      L     #Offset;
      SLD   3;
      LAR2;  // Recupero que offset tiene la String

// --- Ya esta convertido el Valor a ASCI - Fin Patin
CodigoPatin_NUUT_EventosUT:NOP   0;





////////////////////////////////////////////////////////////////////////////////
// --- Atributo de ETIQUETA (Si es necesario) --- Router
      SET;  // Tiene Etiqueta
      AN    "DB850_DefinicionMesas".Mesa[#NumMesa].AtributosGalibo_DeEvento.EtiquetaRouter;
      JC    FinEtiquetaRouter_NUUT_EventoUT;

      OPN   DB [#DBEventos];
      L     '[';  // Evento - Atributo Etiqueta '[SSCC]'
      T     DBB [AR2, P#0.0];
      L     'SSCC';
      T     DBD [AR2, P#1.0];
      L     ']';
      T     DBB [AR2, P#5.0];
      +AR2  P#6.0;

      L     "DB814_UTs_Etiqueta".UT[#NumeroUT].EtiquetaRouter;
      T     #Valor;

// --- Convertir Valor a ASCII -  Etiqueta de Router
      TAR2;
      SRD   3;
      T     #NumBytes;  // Miro que offset tiene la String

      CALL  "FC893_Obtener_StringDelAtributo"
      ( DB_String := #NumDBEventos,
        OffsetIni := #NumBytes,
        Valor     := #Valor,
        OffsetFin := #Offset
      );  // Llamo a ObtenerStrinAtributo

      L     #Offset;
      SLD   3;
      LAR2;  // Recupero que offset tiene la String

// --- Ya esta convertido el Valor a ASCI - Fin Etiqueta de Router
FinEtiquetaRouter_NUUT_EventoUT:NOP   0;





////////////////////////////////////////////////////////////////////////////////
// --- Atributo de ETIQUETA (Si es necesario) ---  STRING
      SET;  // Tiene Etiqueta
      AN    "DB850_DefinicionMesas".Mesa[#NumMesa].AtributosGalibo_DeEvento.EtiquetaString;
      JC    FinEtiquetaString_NUUT_EventoUT;

      OPN   DB [#DBEventos];
      L     '[';  // Evento - Atributo Etiqueta '[SSCC]'
      T     DBB [AR2, P#0.0];
      L     'SSCC';
      T     DBD [AR2, P#1.0];
      L     ']';
      T     DBB [AR2, P#5.0];
      +AR2  P#6.0;

      L     2;  // Puntero a la Etiqueta
      T     #IndiceEtiqueta;

BucleEtiquetastring_NUUT_EventoUT:NOP   0;
      L     "DB814_UTs_Etiqueta".UT[#NumeroUT].Etiqueta[#IndiceEtiqueta];
      T     #Valor;  // Recoge el caracter de la Etiqueta

      L     #Valor;
      L     0;
      ==D;  // Es Final de Etiqueta?
      JC    FinEtiquetaString_NUUT_EventoUT;

      OPN   DB [#DBEventos];
      L     #Valor;
      T     DBB [AR2, P#0.0];

      L     #IndiceEtiqueta;  // Siguiente Caracter
      L     1;
      +I;
      T     #IndiceEtiqueta;
      +AR2  P#1.0;

      JU    BucleEtiquetastring_NUUT_EventoUT;

FinEtiquetaString_NUUT_EventoUT:NOP   0;


////////////////////////////////////////////////////////////////////////////////-
// --- Final del Formato del Evento ---

      OPN   DB [#DBEventos];  // DB de Eventos Generados (A Emitir)
      L     '}';  // Fin de Evento '}'
      T     DBB [AR2, P#0.0];
      +AR2  P#1.0;

////////////////////////////////////////////////////////////////////////////////
////////////////////////////////////////////////////////////////////////////////
////////////////////////////////////////////////////////////////////////////////
////////////////////////////////////////////////////////////////////////////////
// Dar por formateado el Evento
// Borrar la UT de la Base de datos (Por Presencias Multiples de las Mesas)
// Solo no se borra cuando la Mesa es Remota, no debe ni entrar aqui.

      CALL  "FC722_EliminarUT_DeMesa"
      ( NumeroUT := #NumeroUT
      );

      JU    FinBucles_EventosUT;

// Fin del Evento NUUT
////////////////////////////////////////////////////////////////////////////////
////////////////////////////////////////////////////////////////////////////////
////////////////////////////////////////////////////////////////////////////////
////////////////////////////////////////////////////////////////////////////////



NETWORK
TITLE = ---- Evento de UT - Refresco de Datos de la UT -- DATO
GenerarEvento_DATO_EventoUT:NOP   0;

////////////////////////////////////////////////////////////////////////////////
////////////////////////////////////////////////////////////////////////////////
////////////////////////////////////////////////////////////////////////////////
////////////////////////////////////////////////////////////////////////////////
// -- Formateo del Evento DATO - Refresco de Datos de la UT

      L     #P_Eventos;
      LAR2;  // Puntero al DB de Eventos Generados

      TAR2;  // Mirar si es el primer evento de la lista
      L     0;
      ==I;
      JC    InicioBuffer_DATO_EventosUT;  // Es el primero

      OPN   DB [#DBEventos];  // Hay que añadir si no es el primer evento
      L     ',';  // Separador entre eventos ','
      T     DBB [AR2, P#0.0];
      +AR2  P#1.0;

InicioBuffer_DATO_EventosUT:NOP   0;
      OPN   DB [#DBEventos];  // DB de Eventos Generados (A Emitir)
      L     '{';  // Inicio de Evento '{'
      T     DBB [AR2, P#0.0];
      +AR2  P#1.0;

      L     'DATO';  // Evento 'DATO'
      T     DBD [AR2, P#0.0];
      +AR2  P#4.0;


////////////////////////////////////////////////////////////////////////////////
      L     '[';  // Evento - Atributo Mckey '[MCKY]'
      T     DBB [AR2, P#0.0];
      L     'MCKY';
      T     DBD [AR2, P#1.0];
      L     ']';
      T     DBB [AR2, P#5.0];
      +AR2  P#6.0;

      L     "DB812_UTs_Control".UT[#NumeroUT].Mckey;
      T     #Valor;

// --- Convertir Valor a ASCII - Mckey
      TAR2;
      SRD   3;
      T     #NumBytes;  // Miro que offset tiene la String

      CALL  "FC893_Obtener_StringDelAtributo"
      ( DB_String := #NumDBEventos,
        OffsetIni := #NumBytes,
        Valor     := #Valor,
        OffsetFin := #Offset
      );  // Llamo a ObtenerStrinAtributo

      L     #Offset;
      SLD   3;
      LAR2;  // Recupero que offset tiene la String

// --- Ya esta convertido el Valor a ASCI - Fin Mckey


////////////////////////////////////////////////////////////////////////////////
      OPN   DB [#DBEventos];
      L     '[';  // Evento - Atributo Mesa Actual '[MESA]'
      T     DBB [AR2, P#0.0];
      L     'MESA';
      T     DBD [AR2, P#1.0];
      L     ']';
      T     DBB [AR2, P#5.0];
      +AR2  P#6.0;

      L     "DB812_UTs_Control".UT[#NumeroUT].MesaActual;
      T     #Valor;

// --- Convertir Valor a ASCII -  Mesa Actual
      TAR2;
      SRD   3;
      T     #NumBytes;  // Miro que offset tiene la String

      CALL  "FC893_Obtener_StringDelAtributo"
      ( DB_String := #NumDBEventos,
        OffsetIni := #NumBytes,
        Valor     := #Valor,
        OffsetFin := #Offset
      );  // Llamo a ObtenerStrinAtributo

      L     #Offset;
      SLD   3;
      LAR2;  // Recupero que offset tiene la String

// --- Ya esta convertido el Valor a ASCI - Fin Mesa Actual


////////////////////////////////////////////////////////////////////////////////
////////////////////////////////////////////////////////////////////////////////
////////////////////////////////////////////////////////////////////////////////
////////////////////////////////////////////////////////////////////////////////
// --- Caracteristicas de la UT a Emitir


////////////////////////////////////////////////////////////////////////////////
// --- Atributo de ALTURA COTA (Si es necesario) ---
      SET;  // Tiene Cota de Altura ?
      AN    "DB850_DefinicionMesas".Mesa[#NumMesa].AtributosGalibo_DeEvento.Cota_Altura;
      JC    CotaAltura_DATO_EventoUT;

      L     "DB815_UTs_Datos".UT[#NumeroUT].CotaAltura;
      T     #Valor;

      OPN   DB [#DBEventos];
      L     '[';  // Evento - Atributo Altura Cota '[COTA]'
      T     DBB [AR2, P#0.0];
      L     'COTA';
      T     DBD [AR2, P#1.0];
      L     ']';
      T     DBB [AR2, P#5.0];
      +AR2  P#6.0;

// --- Convertir Valor a ASCII -  Altura Cota
      TAR2;
      SRD   3;
      T     #NumBytes;  // Miro que offset tiene la String

      CALL  "FC893_Obtener_StringDelAtributo"
      ( DB_String := #NumDBEventos,
        OffsetIni := #NumBytes,
        Valor     := #Valor,
        OffsetFin := #Offset
      );  // Llamo a ObtenerStrinAtributo

      L     #Offset;
      SLD   3;
      LAR2;  // Recupero que offset tiene la String

// --- Ya esta convertido el Valor a ASCI - Fin Altura Cota
CotaAltura_DATO_EventoUT:NOP   0;


////////////////////////////////////////////////////////////////////////////////
////////////////////////////////////////////////////////////////////////////////
////////////////////////////////////////////////////////////////////////////////
////////////////////////////////////////////////////////////////////////////////
// --- Atributo de GALIBO (Si es necesario) ---
      SET;  // Tiene Altura ?
      AN    "DB850_DefinicionMesas".Mesa[#NumMesa].AtributosGalibo_DeEvento.Altura;
      JC    CodigoAltura_DATO_EventoUT;

      OPN   DB [#DBEventos];
      L     '[';  // Evento - Atributo Galibo Altura '[ALTO]'
      T     DBB [AR2, P#0.0];
      L     'ALTO';
      T     DBD [AR2, P#1.0];
      L     ']';
      T     DBB [AR2, P#5.0];
      +AR2  P#6.0;

      L     "DB815_UTs_Datos".UT[#NumeroUT].GaliboAltura;
      T     #Valor;

// --- Convertir Valor a ASCII -  Alto
      TAR2;
      SRD   3;
      T     #NumBytes;  // Miro que offset tiene la String

      CALL  "FC893_Obtener_StringDelAtributo"
      ( DB_String := #NumDBEventos,
        OffsetIni := #NumBytes,
        Valor     := #Valor,
        OffsetFin := #Offset
      );  // Llamo a ObtenerStrinAtributo

      L     #Offset;
      SLD   3;
      LAR2;  // Recupero que offset tiene la String


// nieves inicio modificación emisión atributo VACI

//Comprobar si tenemos que emitir el evento

      SET;
      L     "DB815_UTs_Datos".UT[#NumeroUT].GaliboVacia;
      L     0;
      ==I;
      JC    CodigoAltura_DATO_EventoUT;

      OPN   DB [#DBEventos];
      L     '[';  // Evento - Atributo Galibo Altura '[ALTO]'
      T     DBB [AR2, P#0.0];
      L     'VACI';
      T     DBD [AR2, P#1.0];
      L     ']';
      T     DBB [AR2, P#5.0];
      +AR2  P#6.0;

      L     "DB815_UTs_Datos".UT[#NumeroUT].GaliboVacia;
      L     1;
      -I;
      T     #Valor;

// --- Convertir Valor a ASCII -  VACIO
      TAR2;
      SRD   3;
      T     #NumBytes;  // Miro que offset tiene la String

      CALL  "FC893_Obtener_StringDelAtributo"
      ( DB_String := #NumDBEventos,
        OffsetIni := #NumBytes,
        Valor     := #Valor,
        OffsetFin := #Offset
      );  // Llamo a ObtenerStrinAtributo


      L     #Offset;
      SLD   3;
      LAR2;  // Recupero que offset tiene la String


// fin modificación atributo VACI

// --- Ya esta convertido el Valor a ASCI - Fin Alto
CodigoAltura_DATO_EventoUT:NOP   0;


////////////////////////////////////////////////////////////////////////////////
      SET;  // Tien Anchura ?
      AN    "DB850_DefinicionMesas".Mesa[#NumMesa].AtributosGalibo_DeEvento.Anchura;
      JC    CodigAnchura_DATO_EventoUT;

      OPN   DB [#DBEventos];
      L     '[';  // Evento - Atributo Galibo Anchura '[ANCH]'
      T     DBB [AR2, P#0.0];
      L     'ANCH';
      T     DBD [AR2, P#1.0];
      L     ']';
      T     DBB [AR2, P#5.0];
      +AR2  P#6.0;

      L     "DB815_UTs_Datos".UT[#NumeroUT].GaliboAnchura;
      T     #Valor;

// --- Convertir Valor a ASCII -  Anchura
      TAR2;
      SRD   3;
      T     #NumBytes;  // Miro que offset tiene la String

      CALL  "FC893_Obtener_StringDelAtributo"
      ( DB_String := #NumDBEventos,
        OffsetIni := #NumBytes,
        Valor     := #Valor,
        OffsetFin := #Offset
      );  // Llamo a ObtenerStrinAtributo

      L     #Offset;
      SLD   3;
      LAR2;  // Recupero que offset tiene la String

// --- Ya esta convertido el Valor a ASCI - Fin Anchura
CodigAnchura_DATO_EventoUT:NOP   0;


////////////////////////////////////////////////////////////////////////////////
      SET;  // Tiene Profundidad ?
      AN    "DB850_DefinicionMesas".Mesa[#NumMesa].AtributosGalibo_DeEvento.Profundidad;
      JC    CodigLargura_DATO_EventoUT;

      OPN   DB [#DBEventos];
      L     '[';  // Evento - Atributo Galibo Profuncidad '[PROF]'
      T     DBB [AR2, P#0.0];
      L     'PROF';
      T     DBD [AR2, P#1.0];
      L     ']';
      T     DBB [AR2, P#5.0];
      +AR2  P#6.0;

      L     "DB815_UTs_Datos".UT[#NumeroUT].GaliboProfundidad;
      T     #Valor;

// --- Convertir Valor a ASCII -  Largura
      TAR2;
      SRD   3;
      T     #NumBytes;  // Miro que offset tiene la String

      CALL  "FC893_Obtener_StringDelAtributo"
      ( DB_String := #NumDBEventos,
        OffsetIni := #NumBytes,
        Valor     := #Valor,
        OffsetFin := #Offset
      );  // Llamo a ObtenerStrinAtributo

      L     #Offset;
      SLD   3;
      LAR2;  // Recupero que offset tiene la String

// --- Ya esta convertido el Valor a ASCI - Fin Largura
CodigLargura_DATO_EventoUT:NOP   0;


////////////////////////////////////////////////////////////////////////////////
      SET;  // Tiene Remontado ?
      AN    "DB850_DefinicionMesas".Mesa[#NumMesa].AtributosGalibo_DeEvento.Remontado;
      JC    CodigRemontado_DATO_EventoUT;

      OPN   DB [#DBEventos];
      L     '[';  // Evento - Atributo Galibo Remontada '[REMO]'
      T     DBB [AR2, P#0.0];
      L     'REMO';
      T     DBD [AR2, P#1.0];
      L     ']';
      T     DBB [AR2, P#5.0];
      +AR2  P#6.0;

      L     "DB815_UTs_Datos".UT[#NumeroUT].GaliboRemontada;
      L     1;
      -I;
      L     W#16#30;
      +I;
      OPN   DB [#DBEventos];
      T     DBB [AR2, P#0.0];
      +AR2  P#1.0;

CodigRemontado_DATO_EventoUT:NOP   0;


////////////////////////////////////////////////////////////////////////////////
// --- Atributo de PESO (Si es necesario) ---
      SET;  // Tiene Peso ?
      AN    "DB850_DefinicionMesas".Mesa[#NumMesa].AtributosGalibo_DeEvento.Peso;
      JC    Peso_DATO_EventoUT;

      OPN   DB [#DBEventos];
      L     '[';  // Evento - Atributo Peso '[PESO]'
      T     DBB [AR2, P#0.0];
      L     'PESO';
      T     DBD [AR2, P#1.0];
      L     ']';
      T     DBB [AR2, P#5.0];
      +AR2  P#6.0;

      L     "DB815_UTs_Datos".UT[#NumeroUT].Peso;
      T     #Valor;

// --- Convertir Valor a ASCII -  Peso
      TAR2;
      SRD   3;
      T     #NumBytes;  // Miro que offset tiene la String

      CALL  "FC893_Obtener_StringDelAtributo"
      ( DB_String := #NumDBEventos,
        OffsetIni := #NumBytes,
        Valor     := #Valor,
        OffsetFin := #Offset
      );  // Llamo a ObtenerStrinAtributo

      L     #Offset;
      SLD   3;
      LAR2;  // Recupero que offset tiene la String

// --- Ya esta convertido el Valor a ASCI - Fin Peso
Peso_DATO_EventoUT:NOP   0;


////////////////////////////////////////////////////////////////////////////////
// --- Atributo de ANCHURA COTA (Si es necesario) ---
      SET;  // Tiene Cota de Anchura ?
      AN    "DB850_DefinicionMesas".Mesa[#NumMesa].AtributosGalibo_DeEvento.Cota_Anchura;
      JC    CotaAnchura_DATO_EventoUT;

      L     "DB815_UTs_Datos".UT[#NumeroUT].CotaAnchura;
      T     #Valor;

      OPN   DB [#DBEventos];
      L     '[';  // Evento - Atributo Anchura Cota '[COTW]'
      T     DBB [AR2, P#0.0];
      L     'COTW';
      T     DBD [AR2, P#1.0];
      L     ']';
      T     DBB [AR2, P#5.0];
      +AR2  P#6.0;

// --- Convertir Valor a ASCII -  Anchura Cota
      TAR2;
      SRD   3;
      T     #NumBytes;  // Miro que offset tiene la String

      CALL  "FC893_Obtener_StringDelAtributo"
      ( DB_String := #NumDBEventos,
        OffsetIni := #NumBytes,
        Valor     := #Valor,
        OffsetFin := #Offset
      );  // Llamo a ObtenerStrinAtributo

      L     #Offset;
      SLD   3;
      LAR2;  // Recupero que offset tiene la String

// --- Ya esta convertido el Valor a ASCI - Fin Anchura Cota
CotaAnchura_DATO_EventoUT:NOP   0;


////////////////////////////////////////////////////////////////////////////////
// --- Atributo de LARGURA COTA (Si es necesario) ---
      SET;  // Tiene Cota de Profundidad ?
      AN    "DB850_DefinicionMesas".Mesa[#NumMesa].AtributosGalibo_DeEvento.Cota_Profundidad;
      JC    CotaLargura_DATO_EventoUT;

      L     "DB815_UTs_Datos".UT[#NumeroUT].CotaProfundidad;
      T     #Valor;

      OPN   DB [#DBEventos];
      L     '[';  // Evento - Atributo Largura Cota '[COTL]'
      T     DBB [AR2, P#0.0];
      L     'COTL';
      T     DBD [AR2, P#1.0];
      L     ']';
      T     DBB [AR2, P#5.0];
      +AR2  P#6.0;

// --- Convertir Valor a ASCII -  Largura Cota
      TAR2;
      SRD   3;
      T     #NumBytes;  // Miro que offset tiene la String

      CALL  "FC893_Obtener_StringDelAtributo"
      ( DB_String := #NumDBEventos,
        OffsetIni := #NumBytes,
        Valor     := #Valor,
        OffsetFin := #Offset
      );  // Llamo a ObtenerStrinAtributo

      L     #Offset;
      SLD   3;
      LAR2;  // Recupero que offset tiene la String

// --- Ya esta convertido el Valor a ASCI - Fin Largura Cota
CotaLargura_DATO_EventoUT:NOP   0;


////////////////////////////////////////////////////////////////////////////////
////////////////////////////////////////////////////////////////////////////////
////////////////////////////////////////////////////////////////////////////////
// --- Atributo de TIPO, HUECO y TACO (Si es necesario) ---
      SET;  // Tiene Taco ?
      AN    "DB850_DefinicionMesas".Mesa[#NumMesa].AtributosGalibo_DeEvento.Taco;
      JC    CodigoTaco_DATO_EventoUT;

      OPN   DB [#DBEventos];
      L     '[';  // Evento - Atributo Galibo Taco '[TACO]'
      T     DBB [AR2, P#0.0];
      L     'TACO';
      T     DBD [AR2, P#1.0];
      L     ']';
      T     DBB [AR2, P#5.0];
      +AR2  P#6.0;

      L     "DB815_UTs_Datos".UT[#NumeroUT].GaliboTaco;
      T     #Valor;

// --- Convertir Valor a ASCII -  Taco
      TAR2;
      SRD   3;
      T     #NumBytes;  // Miro que offset tiene la String

      CALL  "FC893_Obtener_StringDelAtributo"
      ( DB_String := #NumDBEventos,
        OffsetIni := #NumBytes,
        Valor     := #Valor,
        OffsetFin := #Offset
      );  // Llamo a ObtenerStrinAtributo

      L     #Offset;
      SLD   3;
      LAR2;  // Recupero que offset tiene la String

// --- Ya esta convertido el Valor a ASCI - Fin Taco
CodigoTaco_DATO_EventoUT:NOP   0;


////////////////////////////////////////////////////////////////////////////////
      SET;  // Tiene Hueco ?
      AN    "DB850_DefinicionMesas".Mesa[#NumMesa].AtributosGalibo_DeEvento.Hueco;
      JC    CodigoHueco_DATO_EventoUT;

      OPN   DB [#DBEventos];
      L     '[';  // Evento - Atributo Galibo Hueco '[HUEC]'
      T     DBB [AR2, P#0.0];
      L     'HUEC';
      T     DBD [AR2, P#1.0];
      L     ']';
      T     DBB [AR2, P#5.0];
      +AR2  P#6.0;

      L     "DB815_UTs_Datos".UT[#NumeroUT].GaliboHueco;
      T     #Valor;

// --- Convertir Valor a ASCII -  Hueco
      TAR2;
      SRD   3;
      T     #NumBytes;  // Miro que offset tiene la String

      CALL  "FC893_Obtener_StringDelAtributo"
      ( DB_String := #NumDBEventos,
        OffsetIni := #NumBytes,
        Valor     := #Valor,
        OffsetFin := #Offset
      );  // Llamo a ObtenerStrinAtributo

      L     #Offset;
      SLD   3;
      LAR2;  // Recupero que offset tiene la String

// --- Ya esta convertido el Valor a ASCI - Fin Hueco
CodigoHueco_DATO_EventoUT:NOP   0;


////////////////////////////////////////////////////////////////////////////////
      SET;  // Tiene Hueco_R
      AN    "DB850_DefinicionMesas".Mesa[#NumMesa].AtributosGalibo_DeEvento.HuecoRemontado;
      JC    CodigoHuecoR_DATO_EventoUT;

      OPN   DB [#DBEventos];
      L     '[';  // Evento - Atributo Galibo Hueco '[HUEC]'
      T     DBB [AR2, P#0.0];
      L     'HUER';
      T     DBD [AR2, P#1.0];
      L     ']';
      T     DBB [AR2, P#5.0];
      +AR2  P#6.0;

      L     "DB815_UTs_Datos".UT[#NumeroUT].GaliboHuecoRemontado;
      T     #Valor;

// --- Convertir Valor a ASCII -  Hueco R
      TAR2;
      SRD   3;
      T     #NumBytes;  // Miro que offset tiene la String

      CALL  "FC893_Obtener_StringDelAtributo"
      ( DB_String := #NumDBEventos,
        OffsetIni := #NumBytes,
        Valor     := #Valor,
        OffsetFin := #Offset
      );  // Llamo a ObtenerStrinAtributo

      L     #Offset;
      SLD   3;
      LAR2;  // Recupero que offset tiene la String

// --- Ya esta convertido el Valor a ASCI - Fin Hueco R
CodigoHuecoR_DATO_EventoUT:NOP   0;


////////////////////////////////////////////////////////////////////////////////
      SET;  // Tiene Tipo ?
      AN    "DB850_DefinicionMesas".Mesa[#NumMesa].AtributosGalibo_DeEvento.Tipo;
      JC    CodigoTipo_DATO_EventoUT;

      OPN   DB [#DBEventos];
      L     '[';  // Evento - Atributo Galibo Hueco '[HUEC]'
      T     DBB [AR2, P#0.0];
      L     'TIPO';
      T     DBD [AR2, P#1.0];
      L     ']';
      T     DBB [AR2, P#5.0];
      +AR2  P#6.0;

      L     "DB815_UTs_Datos".UT[#NumeroUT].GaliboTipoCarga;
      L     W#16#F;
      <>I;
      JC    CodigoTipoExiste_DATO_EventoUT;

      OPN   DB [#DBEventos];
      L     'ERRO';
      T     DBD [AR2, P#0.0];
      +AR2  P#4.0;

      JU    CodigoTipo_DATO_EventoUT;

CodigoTipoExiste_DATO_EventoUT:NOP   0;
      L     "DB815_UTs_Datos".UT[#NumeroUT].GaliboTipoCarga;
      L     3000;
      +I;
      T     #Convertir;
      CALL  "FC895_Obtener_EtiquetaDeValor"
      ( ValorEvento    := #Convertir,
        EtiquetaEvento := #Conversion
      );

      OPN   DB [#DBEventos];
      L     #Conversion;
      T     DBD [AR2, P#0.0];
      +AR2  P#4.0;

CodigoTipo_DATO_EventoUT:NOP   0;


////////////////////////////////////////////////////////////////////////////////
////////////////////////////////////////////////////////////////////////////////
////////////////////////////////////////////////////////////////////////////////
// --- Atributo de COLOR (Si es necesario) ---
      SET;  // Tiene Color ?
      AN    "DB850_DefinicionMesas".Mesa[#NumMesa].AtributosGalibo_DeEvento.Color;
      JC    CodigoColor_DATO_EventoUT;

      OPN   DB [#DBEventos];
      L     '[';  // Evento - Atributo Galibo Hueco '[HUEC]'
      T     DBB [AR2, P#0.0];
      L     'COLO';
      T     DBD [AR2, P#1.0];
      L     ']';
      T     DBB [AR2, P#5.0];
      +AR2  P#6.0;

      L     "DB815_UTs_Datos".UT[#NumeroUT].GaliboColor;
      L     W#16#F;
      <>I;
      JC    CodigoColorExiste_DATO_EventoUT;

      OPN   DB [#DBEventos];
      L     'ERRO';
      T     DBD [AR2, P#0.0];
      +AR2  P#4.0;

      JU    CodigoColor_DATO_EventoUT;

CodigoColorExiste_DATO_EventoUT:NOP   0;
      L     "DB815_UTs_Datos".UT[#NumeroUT].GaliboColor;
      L     3100;
      +I;
      T     #Convertir;
      CALL  "FC895_Obtener_EtiquetaDeValor"
      ( ValorEvento    := #Convertir,
        EtiquetaEvento := #Conversion
      );

      OPN   DB [#DBEventos];
      L     #Conversion;
      T     DBD [AR2, P#0.0];
      +AR2  P#4.0;

CodigoColor_DATO_EventoUT:NOP   0;

////////////////////////////////////////////////////////////////////////////////
      SET;  // Tiene Patin ?
      AN    "DB850_DefinicionMesas".Mesa[#NumMesa].AtributosGalibo_DeEvento.Patin;
      JC    CodigoPatin_DATO_EventoUT;

      OPN   DB [#DBEventos];
      L     '[';  // Evento - Atributo Galibo Patin '[PATI]'
      T     DBB [AR2, P#0.0];
      L     'PATI';
      T     DBD [AR2, P#1.0];
      L     ']';
      T     DBB [AR2, P#5.0];
      +AR2  P#6.0;

      L     "DB815_UTs_Datos".UT[#NumeroUT].GaliboPatin;
      T     #Valor;

// --- Convertir Valor a ASCII -  Patin
      TAR2;
      SRD   3;
      T     #NumBytes;  // Miro que offset tiene la String

      CALL  "FC893_Obtener_StringDelAtributo"
      ( DB_String := #NumDBEventos,
        OffsetIni := #NumBytes,
        Valor     := #Valor,
        OffsetFin := #Offset
      );  // Llamo a ObtenerStrinAtributo

      L     #Offset;
      SLD   3;
      LAR2;  // Recupero que offset tiene la String

// --- Ya esta convertido el Valor a ASCI - Fin Patin
CodigoPatin_DATO_EventoUT:NOP   0;



////////////////////////////////////////////////////////////////////////////////
// --- Atributo de ETIQUETA (Si es necesario) --- Router
      SET;  // Tiene Etiqueta ?
      AN    "DB850_DefinicionMesas".Mesa[#NumMesa].AtributosGalibo_DeEvento.EtiquetaRouter;
      JC    FinEtiquetaRouter_DATO_EventoUT;

      OPN   DB [#DBEventos];
      L     '[';  // Evento - Atributo Etiqueta '[SSCC]'
      T     DBB [AR2, P#0.0];
      L     'SSCC';
      T     DBD [AR2, P#1.0];
      L     ']';
      T     DBB [AR2, P#5.0];
      +AR2  P#6.0;

      L     0;  // Puntero a la Etiqueta
      T     #IndiceEtiqueta;

      L     "DB814_UTs_Etiqueta".UT[#NumeroUT].EtiquetaRouter;
      T     #Valor;  // Recoge el caracter de la Etiqueta

// --- Convertir Valor a ASCII -  Etiqueta Router
      TAR2;
      SRD   3;
      T     #NumBytes;  // Miro que offset tiene la String

      CALL  "FC893_Obtener_StringDelAtributo"
      ( DB_String := #NumDBEventos,
        OffsetIni := #NumBytes,
        Valor     := #Valor,
        OffsetFin := #Offset
      );  // Llamo a ObtenerStrinAtributo

      L     #Offset;
      SLD   3;
      LAR2;  // Recupero que offset tiene la String

// --- Ya esta convertido el Valor a ASCI - Fin Etiqueta Router
FinEtiquetaRouter_DATO_EventoUT:NOP   0;







////////////////////////////////////////////////////////////////////////////////
// --- Atributo de ETIQUETA (Si es necesario) --- STRING
      SET;  // Tiene Etiqueta ?
      AN    "DB850_DefinicionMesas".Mesa[#NumMesa].AtributosGalibo_DeEvento.EtiquetaString;
      JC    FinEtiquetaString_DATO_EventoUT;

      OPN   DB [#DBEventos];
      L     '[';  // Evento - Atributo Etiqueta '[SSCC]'
      T     DBB [AR2, P#0.0];
      L     'SSCC';
      T     DBD [AR2, P#1.0];
      L     ']';
      T     DBB [AR2, P#5.0];
      +AR2  P#6.0;

      L     2;  // Puntero a la Etiqueta
      T     #IndiceEtiqueta;

BucleEtiquetaString_DATO_EventoUT:NOP   0;
      L     "DB814_UTs_Etiqueta".UT[#NumeroUT].Etiqueta[#IndiceEtiqueta];
      T     #Valor;  // Recoge el caracter de la Etiqueta

      L     #Valor;
      L     0;
      ==I;
      JC    FinEtiquetaString_DATO_EventoUT;  // Es Final de Etiqueta?

      OPN   DB [#DBEventos];
      L     #Valor;
      T     DBB [AR2, P#0.0];

      L     #IndiceEtiqueta;  // Siguiente Caracter
      L     1;
      +I;
      T     #IndiceEtiqueta;
      +AR2  P#1.0;
      JU    BucleEtiquetaString_DATO_EventoUT;

FinEtiquetaString_DATO_EventoUT:NOP   0;





////////////////////////////////////////////////////////////////////////////////
// --- Final del Formato del Evento ---

      OPN   DB [#DBEventos];  // DB de Eventos Generados (A Emitir)
      L     '}';  // Fin de Evento '}'
      T     DBB [AR2, P#0.0];
      +AR2  P#1.0;


////////////////////////////////////////////////////////////////////////////////
////////////////////////////////////////////////////////////////////////////////
////////////////////////////////////////////////////////////////////////////////
////////////////////////////////////////////////////////////////////////////////
// Dar por formateado el Evento

      L     0;  // 0 - Dar por Tratado
      T     "DB812_UTs_Control".UT[#NumeroUT].EstadoEventoAGenerar;

////////////////////////////////////////////////////////////////////////////////
/// Hay que Pedir Datos
      SET;
      AN    "DB812_UTs_Control".UT[#NumeroUT].AtributosDeLaUT.PeticionDeDatos;
      JC    NoPedirDatos_DATO_EventosUT;

      L     141;
      T     "DB812_UTs_Control".UT[#NumeroUT].EstadoEventoAGenerar;

NoPedirDatos_DATO_EventosUT:NOP   0;


////////////////////////////////////////////////////////////////////////////////
      JU    FinBucles_EventosUT;


// Fin del formateo del Evento DATO
////////////////////////////////////////////////////////////////////////////////
////////////////////////////////////////////////////////////////////////////////
////////////////////////////////////////////////////////////////////////////////
////////////////////////////////////////////////////////////////////////////////



NETWORK
TITLE = ---- Evento de UT - Peticion de Datos de la UT - DAT?
GenerarEvento_DAT_EventosUT:NOP   0;

////////////////////////////////////////////////////////////////////////////////
////////////////////////////////////////////////////////////////////////////////
////////////////////////////////////////////////////////////////////////////////
// -- Formateo del Evento DAT? - Peticion de Datos para la UT
// -- Hay que poner que campo?       ¡¡¡ OJO !!!

      L     #P_Eventos;
      LAR2;  // Puntero al DB de Eventos Generados

      TAR2;  // Mirar si es el primer evento de la lista
      L     0;
      ==I;
      JC    InicioBuffer_DAT_EventosUT;  // Es el primero

      OPN   DB [#DBEventos];  // Hay que añadir si no es el primer evento
      L     ',';  // Separador entre eventos ','
      T     DBB [AR2, P#0.0];
      +AR2  P#1.0;

InicioBuffer_DAT_EventosUT:NOP   0;
      OPN   DB [#DBEventos];  // DB de Eventos Generados (A Emitir)
      L     '{';  // Inicio de Evento '{'
      T     DBB [AR2, P#0.0];
      +AR2  P#1.0;

      L     'DAT?';  // Evento 'DAT?'
      T     DBD [AR2, P#0.0];
      +AR2  P#4.0;


////////////////////////////////////////////////////////////////////////////////
      L     '[';  // Evento - Atributo Mckey '[MCKY]'
      T     DBB [AR2, P#0.0];
      L     'MCKY';
      T     DBD [AR2, P#1.0];
      L     ']';
      T     DBB [AR2, P#5.0];
      +AR2  P#6.0;

      L     "DB812_UTs_Control".UT[#NumeroUT].Mckey;
      T     #Valor;

// --- Convertir Valor a ASCII - Mckey
      TAR2;
      SRD   3;
      T     #NumBytes;  // Miro que offset tiene la String

      CALL  "FC893_Obtener_StringDelAtributo"
      ( DB_String := #NumDBEventos,
        OffsetIni := #NumBytes,
        Valor     := #Valor,
        OffsetFin := #Offset
      );  // Llamo a ObtenerStrinAtributo

      L     #Offset;
      SLD   3;
      LAR2;  // Recupero que offset tiene la String

// --- Ya esta convertido el Valor a ASCI - Fin Mckey


////////////////////////////////////////////////////////////////////////////////
      OPN   DB [#DBEventos];
      L     '[';  // Evento - Atributo Mesa Actual '[MESA]'
      T     DBB [AR2, P#0.0];
      L     'MESA';
      T     DBD [AR2, P#1.0];
      L     ']';
      T     DBB [AR2, P#5.0];
      +AR2  P#6.0;

      L     "DB812_UTs_Control".UT[#NumeroUT].MesaActual;
      T     #Valor;

// --- Convertir Valor a ASCII -  Mesa Actual
      TAR2;
      SRD   3;
      T     #NumBytes;  // Miro que offset tiene la String

      CALL  "FC893_Obtener_StringDelAtributo"
      ( DB_String := #NumDBEventos,
        OffsetIni := #NumBytes,
        Valor     := #Valor,
        OffsetFin := #Offset
      );  // Llamo a ObtenerStrinAtributo

      L     #Offset;
      SLD   3;
      LAR2;  // Recupero que offset tiene la String

// --- Ya esta convertido el Valor a ASCI - Fin Mesa Actual


////////////////////////////////////////////////////////////////////////////////
// --- Final del Formato del Evento ---

      OPN   DB [#DBEventos];  // DB de Eventos Generados (A Emitir)
      L     '}';  // Fin de Evento '}'
      T     DBB [AR2, P#0.0];
      +AR2  P#1.0;


////////////////////////////////////////////////////////////////////////////////
////////////////////////////////////////////////////////////////////////////////
////////////////////////////////////////////////////////////////////////////////
////////////////////////////////////////////////////////////////////////////////
// Dar por formateado el Evento

      L     0;  // 0 - Dar por Tratado
      T     "DB812_UTs_Control".UT[#NumeroUT].EstadoEventoAGenerar;

      SET;
      R     "DB812_UTs_Control".UT[#NumeroUT].AtributosDeLaUT.PeticionDeDatos;

      JU    FinBucles_EventosUT;

// Fin del formateo del Evento PD
////////////////////////////////////////////////////////////////////////////////
////////////////////////////////////////////////////////////////////////////////
////////////////////////////////////////////////////////////////////////////////
////////////////////////////////////////////////////////////////////////////////



NETWORK
TITLE = ---- Evento de UT - Chequeo de la UT - CHEQ!
GenerarEvento_CHE_EventosUT:NOP   0;

////////////////////////////////////////////////////////////////////////////////
////////////////////////////////////////////////////////////////////////////////
////////////////////////////////////////////////////////////////////////////////
// -- Formateo del Evento CHE! - Datos UT En Reset
// -- Hay que poner que campo?       ¡¡¡ OJO !!!

      L     #P_Eventos;
      LAR2;  // Puntero al DB de Eventos Generados

      TAR2;  // Mirar si es el primer evento de la lista
      L     0;
      ==I;
      JC    InicioBuffer_CHE_EventosUT;  // Es el primero

      OPN   DB [#DBEventos];  // Hay que añadir si no es el primer evento
      L     ',';  // Separador entre eventos ','
      T     DBB [AR2, P#0.0];
      +AR2  P#1.0;

InicioBuffer_CHE_EventosUT:NOP   0;
      OPN   DB [#DBEventos];  // DB de Eventos Generados (A Emitir)
      L     '{';  // Inicio de Evento '{'
      T     DBB [AR2, P#0.0];
      +AR2  P#1.0;

      L     'CHE!';  // Evento 'DAT?'
      T     DBD [AR2, P#0.0];
      +AR2  P#4.0;


////////////////////////////////////////////////////////////////////////////////
      OPN   DB [#DBEventos];
      L     '[';  // Evento - Atributo TIPO '[TIPO]'
      T     DBB [AR2, P#0.0];
      L     'TIPO';
      T     DBD [AR2, P#1.0];
      L     ']';
      T     DBB [AR2, P#5.0];
      +AR2  P#6.0;

      L     'MCKY';
      T     DBD [AR2, P#0.0];
      +AR2  P#4.0;


////////////////////////////////////////////////////////////////////////////////
      OPN   DB [#DBEventos];
      L     '[';  // Evento - Atributo Mckey '[NUME]'
      T     DBB [AR2, P#0.0];
      L     'NUME';
      T     DBD [AR2, P#1.0];
      L     ']';
      T     DBB [AR2, P#5.0];
      +AR2  P#6.0;

      L     "DB812_UTs_Control".UT[#NumeroUT].Mckey;
      T     #Valor;

// --- Convertir Valor a ASCII - Mckey
      TAR2;
      SRD   3;
      T     #NumBytes;  // Miro que offset tiene la String

      CALL  "FC893_Obtener_StringDelAtributo"
      ( DB_String := #NumDBEventos,
        OffsetIni := #NumBytes,
        Valor     := #Valor,
        OffsetFin := #Offset
      );  // Llamo a ObtenerStrinAtributo

      L     #Offset;
      SLD   3;
      LAR2;  // Recupero que offset tiene la String

// --- Ya esta convertido el Valor a ASCI - Fin Mckey


////////////////////////////////////////////////////////////////////////////////
      OPN   DB [#DBEventos];
      L     '[';  // Evento - Atributo Mesa Actual '[MESA]'
      T     DBB [AR2, P#0.0];
      L     'MESA';
      T     DBD [AR2, P#1.0];
      L     ']';
      T     DBB [AR2, P#5.0];
      +AR2  P#6.0;

      L     "DB812_UTs_Control".UT[#NumeroUT].MesaActual;
      T     #Valor;

// --- Convertir Valor a ASCII -  Mesa Actual
      TAR2;
      SRD   3;
      T     #NumBytes;  // Miro que offset tiene la String

      CALL  "FC893_Obtener_StringDelAtributo"
      ( DB_String := #NumDBEventos,
        OffsetIni := #NumBytes,
        Valor     := #Valor,
        OffsetFin := #Offset
      );  // Llamo a ObtenerStrinAtributo

      L     #Offset;
      SLD   3;
      LAR2;  // Recupero que offset tiene la String

// --- Ya esta convertido el Valor a ASCI - Fin Mesa Actual


////////////////////////////////////////////////////////////////////////////////
      OPN   DB [#DBEventos];
      L     '[';  // Evento - Atributo Resultado '[RESU]'
      T     DBB [AR2, P#0.0];
      L     'RESU';
      T     DBD [AR2, P#1.0];
      L     ']';
      T     DBB [AR2, P#5.0];
      +AR2  P#6.0;

      L     'TRUE';
      T     DBD [AR2, P#0.0];
      +AR2  P#4.0;


////////////////////////////////////////////////////////////////////////////////
// --- Final del Formato del Evento ---

      OPN   DB [#DBEventos];  // DB de Eventos Generados (A Emitir)
      L     '}';  // Fin de Evento '}'
      T     DBB [AR2, P#0.0];
      +AR2  P#1.0;


////////////////////////////////////////////////////////////////////////////////
////////////////////////////////////////////////////////////////////////////////
////////////////////////////////////////////////////////////////////////////////
////////////////////////////////////////////////////////////////////////////////
// Dar por formateado el Evento

      L     0;  // 0 - Dar por Tratado
      T     "DB812_UTs_Control".UT[#NumeroUT].EstadoEventoAGenerar;

      JU    FinBucles_EventosUT;

// Fin del formateo del Evento PD
////////////////////////////////////////////////////////////////////////////////
////////////////////////////////////////////////////////////////////////////////
////////////////////////////////////////////////////////////////////////////////
////////////////////////////////////////////////////////////////////////////////



NETWORK
TITLE = ---- Evento de UT - Peticion de Datos de Embandejado - PEMB // Fecha 07 06 2017
GenerarEvento_PEMB_EventosUT:NOP   0;

////////////////////////////////////////////////////////////////////////////////
////////////////////////////////////////////////////////////////////////////////
///////////////////////////////////////////////////////////////////////////////
// -- Formateo del Evento PEMB (Peticion de Datos de Embandejado de la UT)

      L     #P_Eventos;
      LAR2;  // Puntero al DB de Eventos Generados

      TAR2;  // Mirar si es el primer evento de la lista
      L     0;
      ==I;
      JC    InicioBuffer_PEMB_EventosUT;  // Es el primero

      OPN   DB [#DBEventos];  // Hay que añadir si no es el primer evento
      L     ',';  // Separador entre eventos ','
      T     DBB [AR2, P#0.0];
      +AR2  P#1.0;

InicioBuffer_PEMB_EventosUT:NOP   0;
      OPN   DB [#DBEventos];  // DB de Eventos Generados (A Emitir)
      L     '{';  // Inicio de Evento '{'
      T     DBB [AR2, P#0.0];
      +AR2  P#1.0;

      L     'PEMB';  // Evento 'PEMB'
      T     DBD [AR2, P#0.0];
      +AR2  P#4.0;


////////////////////////////////////////////////////////////////////////////////
      L     '[';  // Evento - Atributo Mckey '[MCKY]'
      T     DBB [AR2, P#0.0];
      L     'MCKY';
      T     DBD [AR2, P#1.0];
      L     ']';  // Evento - Atributo Mckey '[MCKY]'
      T     DBB [AR2, P#5.0];
      +AR2  P#6.0;

      L     "DB812_UTs_Control".UT[#NumeroUT].Mckey;
      T     #Valor;

// --- Convertir Valor a ASCII - Mckey
      TAR2;
      SRD   3;
      T     #NumBytes;  // Miro que offset tiene la String

      CALL  "FC893_Obtener_StringDelAtributo"
      ( DB_String := #NumDBEventos,
        OffsetIni := #NumBytes,
        Valor     := #Valor,
        OffsetFin := #Offset
      );  // Llamo a ObtenerStrinAtributo

      L     #Offset;
      SLD   3;
      LAR2;  // Recupero que offset tiene la String

// --- Ya esta convertido el Valor a ASCI - Fin Mckey


///////////////////////////////////////////////////////////////////////////////
      OPN   DB [#DBEventos];
      L     '[';  // Evento - Atributo Mesa Actual '[MESA]'
      T     DBB [AR2, P#0.0];
      L     'MESA';
      T     DBD [AR2, P#1.0];
      L     ']';
      T     DBB [AR2, P#5.0];
      +AR2  P#6.0;

      L     "DB812_UTs_Control".UT[#NumeroUT].MesaActual;
      T     #Valor;

// --- Convertir Valor a ASCII -  Mesa Actual
      TAR2;
      SRD   3;
      T     #NumBytes;  // Miro que offset tiene la String

      CALL  "FC893_Obtener_StringDelAtributo"
      ( DB_String := #NumDBEventos,
        OffsetIni := #NumBytes,
        Valor     := #Valor,
        OffsetFin := #Offset
      );  // Llamo a ObtenerStrinAtributo

      L     #Offset;
      SLD   3;
      LAR2;  // Recupero que offset tiene la String

// --- Ya esta convertido el Valor a ASCI - Fin Mesa Actual


///////////////////////////////////////////////////////////////////////////////
// --- Final del Formateo del Evento ---

      OPN   DB [#DBEventos];  // DB de Eventos Generados (A Emitir)
      L     '}';  // Fin de Evento '}'
      T     DBB [AR2, P#0.0];
      +AR2  P#1.0;

///////////////////////////////////////////////////////////////////////////////
///////////////////////////////////////////////////////////////////////////////
///////////////////////////////////////////////////////////////////////////////
// Dar por formateado el Evento

      L     0;  // 0 - Dar por Tratado
      T     "DB812_UTs_Control".UT[#NumeroUT].EstadoEventoAGenerar;

      JU    FinBucles_EventosUT;

// Fin del Evento PEMB
///////////////////////////////////////////////////////////////////////////////
///////////////////////////////////////////////////////////////////////////////
///////////////////////////////////////////////////////////////////////////////



NETWORK
TITLE = Generar Eventos de las Mesas
// Recorrer toda las Mesas (Dispositivos)
// Si el Campo EstadoEmision >= 100 se ha generado un evento
EventosMesa:NOP   0;

////////////////////////////////////////////////////////////////////////////////
////////////////////////////////////////////////////////////////////////////////
////////////////////////////////////////////////////////////////////////////////
// - Recorrer todas las Mesas

      L     #InicioBucleMesas;
      T     #NumMesa;

InicioBucle_EventosMesa:NOP   0;
////////////////////////////////////////////////////////////////////////////////
/// Mirar Si pertenece al JDT

      SET;
      X     "DB850_DefinicionMesas".Mesa[#NumMesa].ConfigMesa.MesaDeJDT02;  // JDT01 ?
      XN    #JDT02_Activo;
      =     #MesaDeJDT02;

      SET;
      AN    #MesaDeJDT02;
      JC    ContinuarBucle_EventosMesa;

////////////////////////////////////////////////////////////////////////////////
/// Mirar si esta definido como mesa de Tracking y TL

      SET;
      AN    "DB850_DefinicionMesas".Mesa[#NumMesa].ConfigMesa.MesaPaso;
      AN    "DB850_DefinicionMesas".Mesa[#NumMesa].ConfigMesa.MesaCruce;
      AN    "DB850_DefinicionMesas".Mesa[#NumMesa].ConfigMesa.MesaMultiplesDestinos;
      AN    "DB850_DefinicionMesas".Mesa[#NumMesa].ConfigMesa.MesaTL;
      JC    ContinuarBucle_EventosMesa;


////////////////////////////////////////////////////////////////////////////////

      L     "DB831_Mesas".Mesas[#NumMesa].EstadoEmisionEvento;
      T     #EventoDispositivo;  // Posicion 2

      L     #EventoDispositivo;
      L     100;  // Mirar si hay Evento a Generar
      >=I;  // >= 100 Hay Evento Generado
      JC    Generar_EventosMesa;


////////////////////////////////////////////////////////////////////////////////
// - Continuar con la Suquiente Mesa
ContinuarBucle_EventosMesa:NOP   0;
      L     #NumMesa;  // Si no hay más dispositivos Mesas
      L     #FinalBucleMesas;
      >=I;
      JC    FinalFuncion;  // Ya no hay más dispositivos Mesas, Finalizar

      L     #NumMesa;  // +1, Para la Siguiente Mesa
      L     1;
      +I;
      T     #NumMesa;
      JU    InicioBucle_EventosMesa;

////////////////////////////////////////////////////////////////////////////////
// Comprobacion del tamaño del DB de Eventos Generados
FinBucle_EventosMesa:NOP   0;
      TAR2;
      T     #P_Eventos;
      SRD   3;
      T     #NumBytes;

      L     #NumBytes;  // Miramos si hay sitio
      L     #MaxBytes;
      >I;
      JC    FinalFuncion;  // No se pueden generar más eventos
      JU    ContinuarBucle_EventosMesa;  // Ya se ha generado los eventos de dispositivos mesas



NETWORK
TITLE = Formatear Eventos de las Mesas - Distribucion
// - Distribucion para Eventos de las Mesas
// - Formateo de Eventos
//   - Evento STAT (Cambio de Estado del Dispositivo)
//   - Evento FIN! (Proceso del Dispositivo Finalizado)
//   - Evento DIS? (Pedir datos del Dispositivo)
Generar_EventosMesa:NOP   0;

////////////////////////////////////////////////////////////////////////////////
////////////////////////////////////////////////////////////////////////////////
// -- Formateo del Evento STAT (Estado del Dispositivo)
// -- Formateo del Evento FIN! (Fin del Proceso --> Reset y Paro Blando)
// -- Formateo del Evento DIS? (Peticion de Estado del Dispositivo)
////////////////////////////////////////////////////////////////////////////////
////////////////////////////////////////////////////////////////////////////////
// - Distrubucion de Generarcion de Eventos

      L     #EventoDispositivo;
      L     160;  // Formateo del Evento
      ==I;  // Refresco de datos de la Mesa
      JC    GenerarEvento_STAT_EventosMesa;

      L     #EventoDispositivo;
      L     161;  // Formateo del evento
      ==I;  // Peticion de Datos del Dispositivo
      JC    GenerarEvento_DIS_EventosMesa;

      L     #EventoDispositivo;
      L     151;  // Formateo del Evento
      ==I;  // Fin de Reset OK
      JC    GenerarEvento_FIN_EventosMesa;

      L     #EventoDispositivo;
      L     152;  // Formateo del Evento
      ==I;  // Fin de Reset NOK
      JC    GenerarEvento_FIN_EventosMesa;

      L     #EventoDispositivo;
      L     153;  // Formateo del Evento
      ==I;  // Fin Paro Blando OK
      JC    GenerarEvento_FIN_EventosMesa;

      L     #EventoDispositivo;
      L     154;  // Formateo del Evento
      ==I;  // Fin Paro Blando NOK
      JC    GenerarEvento_FIN_EventosMesa;


////////////////////////////////////////////////////////////////////////////////
////////////////////////////////////////////////////////////////////////////////
// --- Dar por formateado el Evento
// --- No existe el Evento

      L     0;  // Lo doy por tratado
      T     "DB831_Mesas".Mesas[#NumMesa].EstadoEmisionEvento;

      JU    FinBucle_EventosMesa;  // No existe ese tipo de Evento



NETWORK
TITLE = --- Evento de Dispositivo Mesa - Estado de Dispositivo - STAT
////////////////////////////////////////////////////////////////////////////////
////////////////////////////////////////////////////////////////////////////////
////////////////////////////////////////////////////////////////////////////////
// -- Formateo del Evento STAT (Estado del Dispositivo)
GenerarEvento_STAT_EventosMesa:NOP   0;

      L     #P_Eventos;
      LAR2;  // Puntero al DB de Eventos Generados

      TAR2;  // Mirar si es el primer evento de la lista
      L     0;
      ==I;
      JC    InicioBuffer_STAT_EventosMesa;  // Es el primero

      OPN   DB [#DBEventos];
      L     ',';  // Separador entre eventos ','
      T     DBB [AR2, P#0.0];
      +AR2  P#1.0;

InicioBuffer_STAT_EventosMesa:NOP   0;
      OPN   DB [#DBEventos];  // DB de Eventos Generados (A Emitir)
      L     '{';  // Inicio de Evento '{'
      T     DBB [AR2, P#0.0];
      +AR2  P#1.0;

      L     'STAT';  // Evento 'STAT'
      T     DBD [AR2, P#0.0];
      +AR2  P#4.0;


////////////////////////////////////////////////////////////////////////////////
      OPN   DB [#DBEventos];
      L     '[';  // Evento - Atributo Tipo '[TIPO]'
      T     DBB [AR2, P#0.0];
      L     'TIPO';
      T     DBD [AR2, P#1.0];
      L     ']';
      T     DBB [AR2, P#5.0];
      +AR2  P#6.0;

      L     60;  // Dispo Mesa
      T     #Convertir;
      CALL  "FC895_Obtener_EtiquetaDeValor"
      ( ValorEvento    := #Convertir,
        EtiquetaEvento := #Conversion
      );

      OPN   DB [#DBEventos];
      L     #Conversion;
      T     DBD [AR2, P#0.0];
      +AR2  P#4.0;


////////////////////////////////////////////////////////////////////////////////
      L     '[';  // Evento - Atributo Numero de Dispositivo '[NUME]'
      T     DBB [AR2, P#0.0];
      L     'NUME';
      T     DBD [AR2, P#1.0];
      L     ']';
      T     DBB [AR2, P#5.0];
      +AR2  P#6.0;

      L     "CTE_OffsetMesa";
      L     #NumMesa;  // Numero de Mesa
      +I;
      T     #Valor;

// --- Convertir Valor a ASCII - Numero de Mesa
      TAR2;
      SRD   3;
      T     #NumBytes;  // Miro que offset tiene la String

      CALL  "FC893_Obtener_StringDelAtributo"
      ( DB_String := #NumDBEventos,
        OffsetIni := #NumBytes,
        Valor     := #Valor,
        OffsetFin := #Offset
      );  // Llamo a ObtenerStrinAtributo

      L     #Offset;
      SLD   3;
      LAR2;  // Recupero que offset tiene la String

// --- Ya esta convertido el Valor a ASCII


////////////////////////////////////////////////////////////////////////////////
      OPN   DB [#DBEventos];
      L     '[';  // Evento - Atributo Numero de Dispositivo '[NUES]'
      T     DBB [AR2, P#0.0];
      L     'NUES';
      T     DBD [AR2, P#1.0];
      L     ']';
      T     DBB [AR2, P#5.0];
      +AR2  P#6.0;

      L     "DB831_Mesas".Mesas[#NumMesa].StatusActual;
      L     W#16#F;  // Solo la parte Estado
      AW;
      T     #Convertir;

      CALL  "FC895_Obtener_EtiquetaDeValor"
      ( ValorEvento    := #Convertir,
        EtiquetaEvento := #Conversion
      );

      OPN   DB [#DBEventos];
      L     #Conversion;
      T     DBD [AR2, P#0.0];
      +AR2  P#4.0;


////////////////////////////////////////////////////////////////////////////////
      OPN   DB [#DBEventos];
      L     '[';  // Evento - Atributo Numero de Dispositivo '[LLAV]'
      T     DBB [AR2, P#0.0];
      L     'LLAV';
      T     DBD [AR2, P#1.0];
      L     ']';
      T     DBB [AR2, P#5.0];
      +AR2  P#6.0;

      L     "DB831_Mesas".Mesas[#NumMesa].StatusActual;
      L     W#16#F0;  // Solo la parte Llave
      AW;
      SRD   4;
      L     10;
      +I;
      T     #Convertir;

      T     #Convertir;
      CALL  "FC895_Obtener_EtiquetaDeValor"
      ( ValorEvento    := #Convertir,
        EtiquetaEvento := #Conversion
      );

      OPN   DB [#DBEventos];
      L     #Conversion;
      T     DBD [AR2, P#0.0];
      +AR2  P#4.0;


////////////////////////////////////////////////////////////////////////////////
      OPN   DB [#DBEventos];
      L     '[';  // Evento - Atributo Numero de Dispositivo '[HABI]'
      T     DBB [AR2, P#0.0];
      L     'HABI';
      T     DBD [AR2, P#1.0];
      L     ']';
      T     DBB [AR2, P#5.0];
      +AR2  P#6.0;

      L     2001;  // Inicializar: Decir que esta Habilitado
      T     #Convertir;

      SET;
      AN    "DB831_Mesas".Mesas[#NumMesa].Memorias.DesHabilitado;
      JC    HabilitadoDispositivo_STAT_EventosMesa;  // Esta Habilitado ??

      L     2002;
      T     #Convertir;

HabilitadoDispositivo_STAT_EventosMesa:NOP   0;
      CALL  "FC895_Obtener_EtiquetaDeValor"
      ( ValorEvento    := #Convertir,
        EtiquetaEvento := #Conversion
      );

      OPN   DB [#DBEventos];  // Se pasa al Evento
      L     #Conversion;
      T     DBW [AR2, P#0.0];
      +AR2  P#2.0;


////////////////////////////////////////////////////////////////////////////////
      OPN   DB [#DBEventos];
      L     '[';  // Evento - Atributo Numero de Dispositivo '[PRIO]'
      T     DBB [AR2, P#0.0];
      L     'PRIO';
      T     DBD [AR2, P#1.0];
      L     ']';
      T     DBB [AR2, P#5.0];
      +AR2  P#6.0;

      L     "DB831_Mesas".Mesas[#NumMesa].Prioridad;
      T     #Convertir;  // Se pasa a ASCII
      L     W#16#30;
      +I;
      T     #Convertir;

      OPN   DB [#DBEventos];  // Se pasa al Evento
      T     DBB [AR2, P#0.0];
      +AR2  P#1.0;

////////////////////////////////////////////////////////////////////////////////
// Poner Error (Si es necesario)

      L     "DB831_Mesas".Mesas[#NumMesa].ErrorActual;
      L     0;
      ==D;
      JC    SinErrorDispositivo_STAT_EventosMesa;

      L     "DB831_Mesas".Mesas[#NumMesa].ErrorActual;
      T     #Valor;

      OPN   DB [#DBEventos];
      L     '[';  // Evento - Atributo Numero de Dispositivo '[CODE]'
      T     DBB [AR2, P#0.0];
      L     'CODE';
      T     DBD [AR2, P#1.0];
      L     ']';
      T     DBB [AR2, P#5.0];
      +AR2  P#6.0;

// --- Convertir Valor a ASCII - Error
      TAR2;
      SRD   3;
      T     #NumBytes;  // Miro que offset tiene la String

      CALL  "FC893_Obtener_StringDelAtributo"
      ( DB_String := #NumDBEventos,
        OffsetIni := #NumBytes,
        Valor     := #Valor,
        OffsetFin := #Offset
      );  // Llamo a ObtenerStrinAtributo

      L     #Offset;
      SLD   3;
      LAR2;  // Recupero que offset tiene la String

// --- Ya esta convertido el Valor a ASCII

SinErrorDispositivo_STAT_EventosMesa:NOP   0;


////////////////////////////////////////////////////////////////////////////////
// Final del formaateo del Evento

      OPN   DB [#DBEventos];  // DB de Eventos Generados (A Emitir)
      L     '}';  // Fin de Evento '}'
      T     DBB [AR2, P#0.0];
      +AR2  P#1.0;


////////////////////////////////////////////////////////////////////////////////
////////////////////////////////////////////////////////////////////////////////
////////////////////////////////////////////////////////////////////////////////
// Dar por formateado el Evento

      L     0;  // Lo doy por tratado
      T     "DB831_Mesas".Mesas[#NumMesa].EstadoEmisionEvento;

      JU    FinBucle_EventosMesa;  // No existe ese tipo de Evento

// Fin del Formateo del Evento STAT
////////////////////////////////////////////////////////////////////////////////
////////////////////////////////////////////////////////////////////////////////
////////////////////////////////////////////////////////////////////////////////



NETWORK
TITLE = --- Evento de Dispositivo Mesa - Fin de Proceso - FIN!
////////////////////////////////////////////////////////////////////////////////
////////////////////////////////////////////////////////////////////////////////
////////////////////////////////////////////////////////////////////////////////
// -- Formateo del Evento FIN! (Fin del Proceso --> Reset y Paro Blando)
GenerarEvento_FIN_EventosMesa:NOP   0;

      L     #P_Eventos;
      LAR2;  // Puntero al DB de Eventos Generados

      TAR2;  // Mirar si es el primer evento de la lista
      L     0;
      ==I;
      JC    InicioBuffer_FIN_EventosMesa;  // Es el primero

      OPN   DB [#DBEventos];
      L     ',';  // Separador entre eventos ','
      T     DBB [AR2, P#0.0];
      +AR2  P#1.0;

InicioBuffer_FIN_EventosMesa:NOP   0;
      OPN   DB [#DBEventos];  // DB de Eventos Generados (A Emitir)
      L     '{';  // Inicio de Evento '{'
      T     DBB [AR2, P#0.0];
      +AR2  P#1.0;

      L     'FIN!';  // Evento 'FIN!'
      T     DBD [AR2, P#0.0];
      +AR2  P#4.0;


////////////////////////////////////////////////////////////////////////////////
      OPN   DB [#DBEventos];
      L     '[';  // Evento - Atributo Tipo '[TIPO]'
      T     DBB [AR2, P#0.0];
      L     'TIPO';
      T     DBD [AR2, P#1.0];
      L     ']';
      T     DBB [AR2, P#5.0];
      +AR2  P#6.0;

      L     60;  // Dispo Mesa
      T     #Convertir;
      CALL  "FC895_Obtener_EtiquetaDeValor"
      ( ValorEvento    := #Convertir,
        EtiquetaEvento := #Conversion
      );

      OPN   DB [#DBEventos];
      L     #Conversion;
      T     DBD [AR2, P#0.0];
      +AR2  P#4.0;


////////////////////////////////////////////////////////////////////////////////
      L     '[';  // Evento - Atributo Numero de Dispositivo '[NUME]'
      T     DBB [AR2, P#0.0];
      L     'NUME';
      T     DBD [AR2, P#1.0];
      L     ']';
      T     DBB [AR2, P#5.0];
      +AR2  P#6.0;

      L     "CTE_OffsetMesa";
      L     #NumMesa;  // Numero de Mesa
      +I;
      T     #Valor;

// --- Convertir Valor a ASCII - Numero de Maquina
      TAR2;
      SRD   3;
      T     #NumBytes;  // Miro que offset tiene la String

      CALL  "FC893_Obtener_StringDelAtributo"
      ( DB_String := #NumDBEventos,
        OffsetIni := #NumBytes,
        Valor     := #Valor,
        OffsetFin := #Offset
      );  // Llamo a ObtenerStrinAtributo

      L     #Offset;
      SLD   3;
      LAR2;  // Recupero que offset tiene la String

// --- Ya esta convertido el Valor a ASCII


////////////////////////////////////////////////////////////////////////////////
// --- Preparo para los Siguientes Atributos Proceso, Estado del Proceso

      L     22;  // Por defecto Paro Blando
      T     #Proceso;  // Que proceso es

      L     #EventoDispositivo;
      L     153;
      -I;
      T     #ResultadoProceso;  // Resultado del Proceso

      L     #EventoDispositivo;
      L     152;
      >I;
      JC    ParoBlandoProceso_EventosMesa;  // Es Proceso de Paro Balndo ?

      L     21;
      T     #Proceso;  // Que proceso es

      L     #EventoDispositivo;
      L     151;
      -I;
      T     #ResultadoProceso;  // Resultado del Proceso

// --- Continuo con el formateo del evento
ParoBlandoProceso_EventosMesa:NOP   0;


////////////////////////////////////////////////////////////////////////////////
      OPN   DB [#DBEventos];
      L     '[';  // Evento - Atributo Numero de Dispositivo '[PROC]'
      T     DBB [AR2, P#0.0];
      L     'PROC';
      T     DBD [AR2, P#1.0];
      L     ']';
      T     DBB [AR2, P#5.0];
      +AR2  P#6.0;

      L     #Proceso;
      T     #Convertir;

      CALL  "FC895_Obtener_EtiquetaDeValor"
      ( ValorEvento    := #Convertir,
        EtiquetaEvento := #Conversion
      );

      OPN   DB [#DBEventos];
      L     #Conversion;
      T     DBD [AR2, P#0.0];
      +AR2  P#4.0;


////////////////////////////////////////////////////////////////////////////////
      OPN   DB [#DBEventos];
      L     '[';  // Evento - Atributo Numero de Dispositivo '[RSLT]'
      T     DBB [AR2, P#0.0];
      L     'RSLT';
      T     DBD [AR2, P#1.0];
      L     ']';
      T     DBB [AR2, P#5.0];
      +AR2  P#6.0;

      L     #ResultadoProceso;
      L     W#16#30;  // Convertir a ASCII
      +I;

      OPN   DB [#DBEventos];
      T     DBB [AR2, P#0.0];
      +AR2  P#1.0;


////////////////////////////////////////////////////////////////////////////////
// Final del formaateo del Evento

      OPN   DB [#DBEventos];  // DB de Eventos Generados (A Emitir)
      L     '}';  // Fin de Evento '}'
      T     DBB [AR2, P#0.0];
      +AR2  P#1.0;


////////////////////////////////////////////////////////////////////////////////
////////////////////////////////////////////////////////////////////////////////
////////////////////////////////////////////////////////////////////////////////
// Dar por formateado el Evento

      L     0;  // Lo doy por tratado
      T     "DB831_Mesas".Mesas[#NumMesa].EstadoEmisionEvento;

      JU    FinBucle_EventosMesa;  // No existe ese tipo de Evento

// Fin del Formateo del Evento FIN!
////////////////////////////////////////////////////////////////////////////////
////////////////////////////////////////////////////////////////////////////////
////////////////////////////////////////////////////////////////////////////////



NETWORK
TITLE = --- Evento de Dispositivo Mesa - Peticion de Estado del Dipositivo - DIS?
////////////////////////////////////////////////////////////////////////////////
////////////////////////////////////////////////////////////////////////////////
////////////////////////////////////////////////////////////////////////////////
// -- Formateo del Evento DIS? (Peticion de Estado del Dispositivo)
GenerarEvento_DIS_EventosMesa:NOP   0;

      L     #P_Eventos;
      LAR2;  // Puntero al DB de Eventos Generados

      TAR2;  // Mirar si es el primer evento de la lista
      L     0;
      ==I;
      JC    InicioBuffer_DIS_EventosMesa;  // Es el primero

      OPN   DB [#DBEventos];
      L     ',';  // Separador entre eventos ','
      T     DBB [AR2, P#0.0];
      +AR2  P#1.0;

InicioBuffer_DIS_EventosMesa:NOP   0;
      OPN   DB [#DBEventos];  // DB de Eventos Generados (A Emitir)
      L     '{';  // Inicio de Evento '{'
      T     DBB [AR2, P#0.0];
      +AR2  P#1.0;

      L     'DIS?';  // Evento 'DIS?'
      T     DBD [AR2, P#0.0];
      +AR2  P#4.0;


////////////////////////////////////////////////////////////////////////////////
      OPN   DB [#DBEventos];
      L     '[';  // Evento - Atributo Tipo '[TIPO]'
      T     DBB [AR2, P#0.0];
      L     'TIPO';
      T     DBD [AR2, P#1.0];
      L     ']';
      T     DBB [AR2, P#5.0];
      +AR2  P#6.0;

      L     60;  // Dispo Mesa
      T     #Convertir;
      CALL  "FC895_Obtener_EtiquetaDeValor"
      ( ValorEvento    := #Convertir,
        EtiquetaEvento := #Conversion
      );

      OPN   DB [#DBEventos];
      L     #Conversion;
      T     DBD [AR2, P#0.0];
      +AR2  P#4.0;


////////////////////////////////////////////////////////////////////////////////
      L     '[';  // Evento - Atributo Numero de Dispositivo '[NUME]'
      T     DBB [AR2, P#0.0];
      L     'NUME';
      T     DBD [AR2, P#1.0];
      L     ']';
      T     DBB [AR2, P#5.0];
      +AR2  P#6.0;

      L     "CTE_OffsetMesa";
      L     #NumMesa;  // Numero de Mesa
      +I;
      T     #Valor;

// --- Convertir Valor a ASCII - Numero de Mesa
      TAR2;
      SRD   3;
      T     #NumBytes;  // Miro que offset tiene la String

      CALL  "FC893_Obtener_StringDelAtributo"
      ( DB_String := #NumDBEventos,
        OffsetIni := #NumBytes,
        Valor     := #Valor,
        OffsetFin := #Offset
      );  // Llamo a ObtenerStrinAtributo

      L     #Offset;
      SLD   3;
      LAR2;  // Recupero que offset tiene la String

// --- Ya esta convertido el Valor a ASCII


////////////////////////////////////////////////////////////////////////////////
// Final del formaateo del Evento

      OPN   DB [#DBEventos];  // DB de Eventos Generados (A Emitir)
      L     '}';  // Fin de Evento '}'
      T     DBB [AR2, P#0.0];
      +AR2  P#1.0;


////////////////////////////////////////////////////////////////////////////////
////////////////////////////////////////////////////////////////////////////////
////////////////////////////////////////////////////////////////////////////////
// Dar por formateado el Evento

      L     0;  // Lo doy por tratado
      T     "DB831_Mesas".Mesas[#NumMesa].EstadoEmisionEvento;

      JU    FinBucle_EventosMesa;  // No existe ese tipo de Evento

// Fin del Formateo del Evento DIS?
////////////////////////////////////////////////////////////////////////////////
////////////////////////////////////////////////////////////////////////////////
////////////////////////////////////////////////////////////////////////////////



NETWORK
TITLE = Fin de la función
// Se acabo
FinalFuncion:NOP   0;


END_FUNCTION

FUNCTION "FC893_Obtener_StringDelAtributo" : Void   // FC893, LAD
TITLE = "ObtenerStringAtributo" - Convertir a String un Doble Entero
{ S7_Optimized_Access := 'FALSE' }
AUTHOR : TRACKING
NAME : 20130301
VERSION : 3.0
// stored: AutoNumber false, SetENOAutomatically false
   VAR_INPUT
      DB_String : UInt;   // DB donde esta la String
      OffsetIni : UInt;   // Numero de byte de la String donde empieza
      Valor : UDInt;   // Valor a Convertir
   END_VAR
   VAR_OUTPUT
      OffsetFin : UInt;   // Numero de byte de la String donde acaba
   END_VAR
   VAR_TEMP
      PunteroDB : DWord;   // Puntero al DB de la String
      NumDB : Word;   // Num. del DB de la String
      ValorRestante : UDInt;   // Valor a convertir que va quedando
      OffsetActual : UInt;   // Numero de byte que estoy desplazando de la String
      Digito : UInt;   // Valor Convertiodo a Guardar en la String
      Temporal : UInt;
      TEMP_OffsetFin : UInt;
   END_VAR
BEGIN

NETWORK
TITLE = Inicializaciones
// Inicializar las Variables que se necesitan
      L     #Valor;  // Inicializo el Valor a Convertir
      T     #ValorRestante;

      L     #DB_String;
      T     #NumDB;

      L     #OffsetIni;  // Apunta al primer caracter el de Mayor peso
      T     #OffsetActual;
      T     #TEMP_OffsetFin;



NETWORK
TITLE = Conversion
// - Mirar si queda numero a convertir
// - Coger digito
// - Guardarlo en la String
// - Conseguir el Valor Restante
InicioBucle:NOP   0;

// -----------------------------------------------------------------------------------------------
// Coger el digito que necesitamos porner en la String - Menor peso

      L     #ValorRestante;
      L     10;
      MOD;  // Obtenemos el digito
      L     W#16#30;  // Y lo convertimos a Char
      +I;  // Sumar W#16#30
      T     #Digito;


// -----------------------------------------------------------------------------------------------
// Guardarlo en la String

      OPN   DB [#NumDB];

      L     #OffsetIni;  // Miro si es el Primer digito
      L     #TEMP_OffsetFin;
      ==I;
      JC    FinalDesplazar;  // Lo es

// Despalzar en la String para meter un nuevo digito

      L     #TEMP_OffsetFin;  // Inicializo al final
      T     #OffsetActual;  // Primer destino del desplazamiento
InicioDesPlazar:L     #OffsetActual;  // Recogo el dato del Byte Origen
      L     1;
      -I;
      SLD   3;
      T     #PunteroDB;
      L     DBB [#PunteroDB];
      T     #Temporal;

      L     #OffsetActual;  // Dejo el dato del Byte Destino
      SLD   3;
      T     #PunteroDB;
      L     #Temporal;
      T     DBB [#PunteroDB];

      L     #OffsetActual;  // Quito un digito para pasra el Siguiente
      L     1;
      -I;
      T     #OffsetActual;

      L     #OffsetActual;  // Se mira si estan todos desplazados
      L     #OffsetIni;
      ==I;
      JC    FinalDesplazar;  // Si estan todos
      JU    InicioDesPlazar;

// Guardo el ultimo digito guardado - Es el más significativo por ahora

FinalDesplazar:L     #OffsetIni;  // Guardo el digito convertido
      SLD   3;
      T     #PunteroDB;
      L     #Digito;
      T     DBB [#PunteroDB];

      L     #TEMP_OffsetFin;  // Incremento el Puntero Final de la String
      L     1;
      +I;
      T     #TEMP_OffsetFin;

// -----------------------------------------------------------------------------------------------
// Conseguimos el Valor Restante

      L     #ValorRestante;  // Dividimos en 10 para sacar el nuevo valor
      L     10;
      /D;
      T     #ValorRestante;

// -----------------------------------------------------------------------------------------------
// Mirar si queda nuero a convertir

      L     #ValorRestante;  // Validamos de que se trata de un numero
      L     0;  // No debe ser: Valor Restante < 0
      <=D;
      JC    Final;  // Se acabado el numero

      JU    InicioBucle;  // Vamos a ver si hay más digitos



NETWORK
TITLE = Final
// Final de la Funcion
Final:NOP   0;

      L     #TEMP_OffsetFin;  // - Devuelvo el Offset Temporal
      T     #OffsetFin;


END_FUNCTION

FUNCTION "FC722_EliminarUT_DeMesa" : Void   // FC722, LAD
TITLE = EliminarUT_DeMesa - Eliminar la UT de la BD
{ S7_Optimized_Access := 'FALSE' }
AUTHOR : TRACKING
NAME : 20130301
VERSION : 3.0
// stored: AutoNumber false, SetENOAutomatically false
   VAR_INPUT
      NumeroUT : UInt;
   END_VAR
   VAR_TEMP
      Mesa : UInt;   // Mesa
      AnteriorUT : UInt;   // UT Anterior
      SiguienteUT : UInt;   // UT Siguiente
      MckeyTemporal : UDInt;   // Para la ordenacion con Mckey
      ColaMckey : UInt;
      ValorReturn : Int;
      Cero : Byte;
   END_VAR
BEGIN

NETWORK
TITLE = Inicilizar
////////////////////////////////////////////////////////////////////////////////
////////////////////////////////////////////////////////////////////////////////
// Inicializa las variables
      L     0;
      T     #AnteriorUT;
      T     #SiguienteUT;



NETWORK
TITLE = Modificar BD de la Mesa -- Previo
////////////////////////////////////////////////////////////////////////////////
////////////////////////////////////////////////////////////////////////////////
////////////////////////////////////////////////////////////////////////////////
// Datos de la UT Mesa, Anterior UT y Siguiente UT
      L     "DB812_UTs_Control".UT[#NumeroUT].MesaActual;
      L     "CTE_OffsetMesa";
      -I;
      T     #Mesa;

      L     "DB812_UTs_Control".UT[#NumeroUT].UT_AnteriorMesa;
      T     #AnteriorUT;
      L     "DB812_UTs_Control".UT[#NumeroUT].UT_SiguienteMesa;
      T     #SiguienteUT;

      L     "DB812_UTs_Control".UT[#NumeroUT].Mckey;
      T     #MckeyTemporal;



////////////////////////////////////////////////////////////////////////////////
// Limpieza de la UT

      L     0;  // Valor a rellenar
      T     #Cero;

// Borrado del DB de los Datos de la UT
      CALL  FILL
      ( BVAL    := #Cero,
        RET_VAL := #ValorReturn,
        BLK     := "DB812_UTs_Control".UT[#NumeroUT]
      );

// Borrado del DB de la Rutas de la UT
      CALL  FILL
      ( BVAL    := #Cero,
        RET_VAL := #ValorReturn,
        BLK     := "DB813_UTs_Ruta".UT[#NumeroUT]
      );

// Borrado del DB de los Datos Auxiliares de la UT
      CALL  FILL
      ( BVAL    := #Cero,
        RET_VAL := #ValorReturn,
        BLK     := "DB814_UTs_Etiqueta".UT[#NumeroUT]
      );
      CALL  FILL
      ( BVAL    := #Cero,
        RET_VAL := #ValorReturn,
        BLK     := "DB815_UTs_Datos".UT[#NumeroUT]
      );
      CALL  FILL
      ( BVAL    := #Cero,
        RET_VAL := #ValorReturn,
        BLK     := "DB816_UTs_TextoPantalla".UT[#NumeroUT]
      );
      CALL  FILL
      ( BVAL    := #Cero,
        RET_VAL := #ValorReturn,
        BLK     := "DB820_UTs_DatosQUBIQA".UT[#NumeroUT]
      );
      CALL  FILL
      ( BVAL    := #Cero,
        RET_VAL := #ValorReturn,
        BLK     := "DB821_UTs_DatosIKPAL".UT[#NumeroUT]
      );



NETWORK
TITLE = -- UT Anterior
////////////////////////////////////////////////////////////////////////////////
////////////////////////////////////////////////////////////////////////////////
////////////////////////////////////////////////////////////////////////////////
// Modificar la UT Anterior
      SET;
      L     #AnteriorUT;
      L     0;
      ==I;  // Era la UT primera de la Mesa
      JC    PrimeraUT_EnColaMesa;
      JU    NoPrimeraUT_EnColaMesa;


////////////////////////////////////////////////////////////////////////////////
// No es la primar UT de la Mesa
NoPrimeraUT_EnColaMesa:NOP   0;
      L     #SiguienteUT;
      T     "DB812_UTs_Control".UT[#AnteriorUT].UT_SiguienteMesa;

      JU    SiguienteUT_EnColaMesa;


////////////////////////////////////////////////////////////////////////////////
// Es la primera UT de la Mesa
PrimeraUT_EnColaMesa:NOP   0;
      L     #SiguienteUT;
      T     "DB810_ColasMesas".Colas[#Mesa].UT_PrimeraMesa;

      JU    SiguienteUT_EnColaMesa;



NETWORK
TITLE = -- UT Siguiente
////////////////////////////////////////////////////////////////////////////////
////////////////////////////////////////////////////////////////////////////////
////////////////////////////////////////////////////////////////////////////////
// Modificar la UT Siguiente
SiguienteUT_EnColaMesa:NOP   0;
      L     #SiguienteUT;
      L     0;
      ==I;
      JC    Final_EnColaDeMesa;  // Era la UT ultima de la Mesa

////////////////////////////////////////////////////////////////////////////////
// No es la Ultima UT de la Mesa
      L     #AnteriorUT;
      T     "DB812_UTs_Control".UT[#SiguienteUT].UT_AnteriorMesa;

      JU    Final_EnColaDeMesa;



NETWORK
TITLE = -- Final
////////////////////////////////////////////////////////////////////////////////
////////////////////////////////////////////////////////////////////////////////
////////////////////////////////////////////////////////////////////////////////
Final_EnColaDeMesa:NOP   0;



NETWORK
TITLE = Modificar BD de la Ordenacion del Mckey -- Previo
////////////////////////////////////////////////////////////////////////////////
////////////////////////////////////////////////////////////////////////////////
////////////////////////////////////////////////////////////////////////////////
// ----- Antes de acabar eliminar de la ordenacion por Mckey

      L     0;  // Si Mckey es 0
      L     #MckeyTemporal;  // Nunca se ha ordenado por Mckey
      ==D;
      JC    Final_EnColaMckey;  // Ir al final de la ordenacion por Mckey


////////////////////////////////////////////////////////////////////////////////
////////////////////////////////////////////////////////////////////////////////
////////////////////////////////////////////////////////////////////////////////
      L     #MckeyTemporal;
      L     10000;  // Hay 10.000 Colas para el Mckey
      MOD;
      T     #ColaMckey;  // Numero de la Cola del Mckey


      L     "DB811_ColasMckeys".MckeyUT[#NumeroUT].UT_AnteriorMckey;
      T     #AnteriorUT;
      L     "DB811_ColasMckeys".MckeyUT[#NumeroUT].UT_SiguienteMcKey;
      T     #SiguienteUT;

// Limpieza
      L     0;
      T     "DB811_ColasMckeys".MckeyUT[#NumeroUT].UT_AnteriorMckey;
      T     "DB811_ColasMckeys".MckeyUT[#NumeroUT].UT_SiguienteMcKey;



NETWORK
TITLE = -- UT Anterior
////////////////////////////////////////////////////////////////////////////////
////////////////////////////////////////////////////////////////////////////////
////////////////////////////////////////////////////////////////////////////////
// ----- UT Anterior Mckey
      L     #AnteriorUT;
      L     0;
      ==I;  // Esta la primera ??????
      JC    PrimeraUT_EnColaMckey;
      JU    NoPrimeraUT_EnColaMckey;


////////////////////////////////////////////////////////////////////////////////
// ----- No es la primera
NoPrimeraUT_EnColaMckey:NOP   0;
      L     #SiguienteUT;
      T     "DB811_ColasMckeys".MckeyUT[#AnteriorUT].UT_SiguienteMcKey;

      JU    SiguienteUT_EnColaMckey;  // Ir a ordenar la UT siguiente


////////////////////////////////////////////////////////////////////////////////
// ------ Es la Pimera
PrimeraUT_EnColaMckey:NOP   0;
      L     #SiguienteUT;
      T     "DB811_ColasMckeys".Colas_Mckey[#ColaMckey].UT_PrimerMckey;

      JU    SiguienteUT_EnColaMckey;  // Ir a Ordenar la UT siguinete



NETWORK
TITLE = -- UT Siguiente
////////////////////////////////////////////////////////////////////////////////
////////////////////////////////////////////////////////////////////////////////
////////////////////////////////////////////////////////////////////////////////
// ---- UT Siguinete Mckey
SiguienteUT_EnColaMckey:NOP   0;
      L     #SiguienteUT;
      L     0;
      ==I;
      JC    Final_EnColaMckey;  // Esta la ultima ????


////////////////////////////////////////////////////////////////////////////////
/// ---- No ses la Ultima
      L     #AnteriorUT;
      T     "DB811_ColasMckeys".MckeyUT[#SiguienteUT].UT_AnteriorMckey;

      JU    Final_EnColaMckey;  // Ir al final de la ordenacion por Mckey



NETWORK
TITLE = -- Final
////////////////////////////////////////////////////////////////////////////////
////////////////////////////////////////////////////////////////////////////////
////////////////////////////////////////////////////////////////////////////////
// Se acabo la ordenacion

Final_EnColaMckey:NOP   0;




END_FUNCTION

FUNCTION "FC805_JDT01AnalisisEnviados" : Void   // FC805, LAD
TITLE = "AnalisisEnviados" - Prepara el Mensaje KA o Lista de Eventos
{ S7_Optimized_Access := 'FALSE' }
AUTHOR : TRACKING
NAME : 20160525
VERSION : 4.1
// - Inicilizar
// - Distribucion
// - Reenviar Mensaje Anterior
// - Emitir Mensaje PING - Keep Alive
// - Emitir Nueva Lista de Eventos
// stored: AutoNumber false, SetENOAutomatically false
   VAR_TEMP
      DBUltimoEmi : Word;   // Num. DB del Ultimo Mensaje Emitido
      DBEventosEmi : Word;   // Num. DB de la Lista de Eventos Generados (Emitir)
      Longitud : UDInt;
      Valor : Int;
      IdentEmisor : DInt;
      IdentReceptor : DInt;
      TMPEsperaAK : UDInt;
      TMPEnvioKA : UDInt;
   END_VAR
BEGIN

NETWORK
TITLE = Inicilizar
// - Inicializar Variables de los DB's
// - Coger de la configuracion el Identificador del Emisor (12)
// - Coger de la configuracion el Identificador del Receptor (18)
// - Temporizador de Espera ACKN - Confirmacion
// - Temporizador de Emision PING - Keep Alive
// - Mirar si el enlace esta activo
// -------------------------------------------------------------------------------------------
// Si trabaja sin Agencia  2016 05 25
      SET;
      A     "Activar_JDT01";  // Mirar si se trabaja con agencia
      JC    ExisteAngencia;

// Solo Borrar si hay algo
      L     "DB808_JDT01EventosGenerados".Mensaje[0];
      L     0;
      ==I;
      JC    Final;

      CALL  "FC898_BorrarMensaje"
      ( DB_A_RESET := "DB808_JDT01EventosGenerados"  // ¿Hay que borrarlo asi?
      );  // Damos por acabado EventosGenerados

      JU    Final;  // Se ha finalizado

ExisteAngencia:NOP   0;

// -------------------------------------------------------------------------------------------
// Inicializar Variables de los DB's

      L     "JDT1_NDB_UltimoEmi";  // Cogemos el DB de UltimoEnviado
      T     #DBUltimoEmi;
      L     "JDT1_NDB_EventosEmi";  // Cogemos el DB de EventosGenerados
      T     #DBEventosEmi;


// --------------------------------------------------------------------------------------------
// Coger de la configuracion el Idendificador del emisor

      L     "JDT1_IdentEmisor";
      T     #IdentEmisor;

// --------------------------------------------------------------------------------------------
// Coger de la configuracion el Idendificador del receptor

      L     "JDT1_IdentReceptor";
      T     #IdentReceptor;

// -------------------------------------------------------------------------------------------
// Mirar si el enlace esta activo

      AN    "DB801_JDT01StatusCOM".EnlaceCP_OK;
      JC    Final;  // El EnlaceCP esta NOK, no hacer nada

// -------------------------------------------------------------------------------------------
// Temporizador de Espera PING - Confirmacion del Mensaje enviado, para el reenvio de Mensaje

      L     "JDT1_TMPEsperaAK";
      T     #TMPEsperaAK;
      CALL  "FC899_TMP"
      ( Temporizar     := "DB801_JDT01StatusCOM".EsperandoAK,
        Valor_Tiempo   := #TMPEsperaAK,  // Tiempo de 10 Segundos
        Base_tiempo_ms := 1000,
        Tiempo_OK      := "DB801_JDT01StatusCOM".TMPEsperaAK_OK,
        Valor_Actual   := "DB801_JDT01StatusCOM".TMPEsperaAK
      );

// -------------------------------------------------------------------------------------------
// Temporizador de Emision PING - Keep Alive (Si no hay actividad)

      L     "JDT1_TMPEnvioKA";
      T     #TMPEnvioKA;
      CALL  "FC899_TMP"
      ( Temporizar     := "DB801_JDT01StatusCOM".SinActividad,
        Valor_Tiempo   := #TMPEnvioKA,  // Tiempo de 1 Minuto
        Base_tiempo_ms := 1000,
        Tiempo_OK      := "DB801_JDT01StatusCOM".TMPEnvioKA_OK,
        Valor_Actual   := "DB801_JDT01StatusCOM".TMPEnvioKA
      );


NETWORK
TITLE = Distribucion
// - Miro si el mensaje anterior esta enviado correctamente
// - Mirar si es mensaje de lista de eventos, para tener que reenvialo
// - Miramos si Hay que Emitir Lista de Eventos
// - Miramos si ha pasado el tiempo para emitir el mensaje PING - Keep Alive
// -------------------------------------------------------------------------------------------
// 1º Paso - Miro si el mensaje anterior esta enviado correctamente
      L     0;
      LAR1;
      OPN   DB [#DBUltimoEmi];
      L     DBB [AR1, P#0.0];
      L     0;
      ==I;  // Esta Tratado el mensaje anterior
      JC    SiguienteMensaje;  // Ir a tratar el siguiente

// -------------------------------------------------------------------------------------------
// 2º Paso - No esta libre. Hay que ver si el Anterior Mensaje es de Lista de eventos
//           Para ver si hay que reenviar el Mensaje

      OPN   DB [#DBUltimoEmi];
      L     DBB [AR1, P#0.0];
      L     'N';  // Si tiene 'N' es un Mensaje de Lista de Eventos
      ==I;
      JC    EmisionEvento_ReEnviar;  // Ir Emitir Reenvio del Evento si es necesario

      SET;  // No se ha emitido todavia
      R     "DB801_JDT01StatusCOM".EsperandoAK;
      JU    Final;  // No hay nada todavia

// -------------------------------------------------------------------------------------------
// 3º Paso - Esta libre. Miramos si Hay que Emitir Lista de Eventos

SiguienteMensaje:L     0;  // Mirar si hay Lista de Eventos a Emitir
      LAR1;
      OPN   DB [#DBEventosEmi];
      L     DBB [AR1, P#0.0];
      L     '{';
      ==I;
      JC    EmisionEvento_ListaDeEventos;  // Ir a Emitir Nueva Lista de Eventos

// -------------------------------------------------------------------------------------------
// 4º Paso - No hay actividad. Miramos si ha pasado el tiempo para emitir el mensaje KA
      SET;
      S     "DB801_JDT01StatusCOM".SinActividad;

      A     "DB801_JDT01StatusCOM".TMPEnvioKA_OK;
      JC    EmisionEvento_KeepAlive;  // Ir a Emitir el Mensaje KA

      JU    Final;  // No va hacerse nada por ahora




NETWORK
TITLE = Reenvio del Mensaje Anterior
// - Mirar si ha pasaso el Tiempo de Espera del Mensaje ACKN - Confirmacion
// - Reenviar el Mensaje Anterior
EmisionEvento_ReEnviar:NOP   0;

// -------------------------------------------------------------------------------------------
// 1º Paso - Mirar si ha pasado el tiempo de Espera del Mensaje AK - Confirmacion

      SET;
      S     "DB801_JDT01StatusCOM".EsperandoAK;

      AN    "DB801_JDT01StatusCOM".TMPEsperaAK_OK;
      JC    Final;

// -------------------------------------------------------------------------------------------
// Reeenviar el mensaje anterior
// Solo Cambiar el primer digito 'N' -> 0x02

//Nieves 26/05/25 Control de los reintentos

// evaluamos si ya hemos intentado emitir el mensaje 3 veces
      SET;
      L     "Reintentos_JDT1";
      L     3;
      <=I;
      JC    reintenta;

// si ya hemos llegado a 3 reintentos, forzamos la desconexión

      L     1;
      T     "Reintentos_JDT1";
      SET;
      S     "DB801_JDT01StatusCOM".EmiJdT_Reset;
      JU    Final;  // Se ha finalizado

reintenta:NOP   0;
      L     "Reintentos_JDT1";
      L     1;
      +I;
      T     "Reintentos_JDT1";



// fin control reintentos

      SET;  // Voy ha Reenviar el Mensaje
      R     "DB801_JDT01StatusCOM".EsperandoAK;  // Con esto reseto el timer

      L     0;
      LAR1;
      OPN   DB [#DBUltimoEmi];  // Cambio el inicio del Mensaje
      L     2;
      T     DBB [AR1, P#0.0];




      JU    Final;  // Se ha finalizado


NETWORK
TITLE = Emitir PING - Keep Alive
// - Resetear variables
// - Formateo del Mensaje PING - Keep Alive
EmisionEvento_KeepAlive:NOP   0;
      O;
// -------------------------------------------------------------------------------------------
// 1º Paso - Resetear variables

      SET;  // Si hay Actividad
      R     "DB801_JDT01StatusCOM".SinActividad;  // Con esto reseto el timer

// -------------------------------------------------------------------------------------------
// 2º Paso - Formateo en Mensaje KA - Con el ultimo secuencial

// Numero Secuencial - Con el ultimo secuencial

      CALL  "FC891_EtiqDInt_EtiqChar"
      ( DB_String   := "JDT1_NDB_UltimoEmi",  // DB UltimoEmision
        Long_String := 4,
        Offset_Ini  := 4,
        Valor       := "DB801_JDT01StatusCOM".ID_UltimoEnviado
      );  // Rellenar el ID del Mensaje

      L     0;  // Puntero DB UltimoEmision
      LAR1;
      OPN   DB [#DBUltimoEmi];

      L     2;  // Primer Byte 0x02 - Para que sea enviada
      T     DBB [AR1, P#0.0];
      L     ';';  // Separador
      T     DBB [AR1, P#5.0];

      L     #IdentEmisor;  // Rellenar el Campo Emisor
      T     DBD [AR1, P#6.0];

      L     ';';  // Separador
      T     DBB [AR1, P#10.0];

      L     #IdentReceptor;  // Rellenar el Campo Receptor
      T     DBD [AR1, P#11.0];

      L     ';';  // Separador
      T     DBB [AR1, P#15.0];

      L     '0';  // Campo Tamaño del Mensaje
      T     DBB [AR1, P#16.0];  // En dos partes '0' y '0031'
      L     '0031';
      T     DBD [AR1, P#17.0];

      L     ';';  // Separador
      T     DBB [AR1, P#21.0];

// Evento  a escrribir- ({KA})

      L     '({';  // Empieza Evento
      T     DBW [AR1, P#22.0];
      L     'PING';  // Evento AK
      T     DBD [AR1, P#24.0];
      L     '})';  // Final del Evento
      T     DBW [AR1, P#28.0];

      L     3;  // Final del Mensaje 0x03
      T     DBB [AR1, P#30.0];

      JU    Final;  // Se ha finalizado


NETWORK
TITLE = Emitir Nueva Lista de Eventos
// - Obtener nuevo numero secuencial
// - Formateo de la Cabecera del Mensaje
// - Formateo del Cuerpo del Mensaje - Lista de Eventos
// - Formateo el final del Mensaje
EmisionEvento_ListaDeEventos:NOP   0;

// -------------------------------------------------------------------------------------------
// 1º Paso - Obtener nuevo numero secuencial

      L     "DB801_JDT01StatusCOM".ID_UltimoEnviado;
      L     1;  // Se Suma +1
      +D;
      T     "DB801_JDT01StatusCOM".ID_UltimoEnviado;  // Guardo el Nuevo ID

      L     "DB801_JDT01StatusCOM".ID_UltimoEnviado;
      L     9999;  // Ha pasado el Limite
      <=I;
      JC    _050;

      L     1;  // Empieza de nuevo
      T     "DB801_JDT01StatusCOM".ID_UltimoEnviado;  // Guardo el Nuevo ID

_050: L     "DB801_JDT01StatusCOM".ID_UltimoEnviado;
      T     #Valor;  // Valor del ID del Mensaje

// -------------------------------------------------------------------------------------------
// 2º Paso -  Formateo de la Cabecera del Mensaje
// Nota: Faltara el tamaño del mensaje que se hara al final

      CALL  "FC891_EtiqDInt_EtiqChar"
      ( DB_String   := "JDT1_NDB_UltimoEmi",  // DB UltimoEmision
        Long_String := 4,
        Offset_Ini  := 4,
        Valor       := "DB801_JDT01StatusCOM".ID_UltimoEnviado
      );  // Rellenar el ID del Mensaje

      L     0;  // Puntero DB UltimoEmision
      LAR1;

      OPN   DB [#DBUltimoEmi];
      L     2;  // Primer Byte 0x02 - Para que sea enviada
      T     DBB [AR1, P#0.0];
      L     ';';  // Separador
      T     DBB [AR1, P#5.0];


      L     #IdentEmisor;  // Rellenar el Campo Emisor
      T     DBD [AR1, P#6.0];

      L     ';';  // Separador
      T     DBB [AR1, P#10.0];

      L     #IdentReceptor;  // Rellenar el Campo Receptor
      T     DBD [AR1, P#11.0];

      L     ';';  // Separador
      T     DBB [AR1, P#15.0];

// Falta el tamaño que se rellenara con el final

      L     ';';  // Separador
      T     DBB [AR1, P#21.0];

      L     '(';  // Inicio de la Lista de Eventos
      T     DBB [AR1, P#22.0];

// -------------------------------------------------------------------------------------------
// 3º Paso -  Formateo del Cuerpo del Mensaje - Lista de Eventos

      +AR1  P#23.0;  // AR1 = PunteroDestino
      L     0;  // AR2 = PunteroOrigen
      LAR2;

_051: OPN   DB [#DBEventosEmi];  // Transferir los datos
      L     DBB [AR2, P#0.0];  // De Origen
      OPN   DB [#DBUltimoEmi];
      T     DBB [AR1, P#0.0];  // A Destino

      L     0;  // Si es 0 - Ha llegado al final de la lista de Eventos
      ==I;
      JC    _052;  // Si Ha llegado al final

      +AR1  P#1.0;  // Se incrementa los punteros
      +AR2  P#1.0;
      JU    _051;

// -------------------------------------------------------------------------------------------
// 4º Paso -  Formateo del Final del Mensaje

_052: OPN   DB [#DBUltimoEmi];
      L     ')';  // Final de la Lista de Eventos
      T     DBB [AR1, P#0.0];

      L     3;  // Ultimo Byte - 0x03
      T     DBB [AR1, P#1.0];

// -------------------------------------------------------------------------------------------
// 5º Paso - Poner el tamaño del Mensaje

      TAR1;  // Calculo el Tamaño del Mensaje
      SRD   3;
      L     2;  // Añadir los dos ultimos digitos
      +D;
      T     #Longitud;

      CALL  "FC891_EtiqDInt_EtiqChar"
      ( DB_String   := "JDT1_NDB_UltimoEmi",  // DB UltimoEmision
        Long_String := 5,
        Offset_Ini  := 20,
        Valor       := #Longitud
      );  // Rellenar el Campo Tamaño del mensaje

// -------------------------------------------------------------------------------------------
// 6º Paso - Limpio las variables

      SET;
      S     "DB801_JDT01StatusCOM".EsperandoAK;

      CALL  "FC898_BorrarMensaje"
      ( DB_A_RESET := "DB808_JDT01EventosGenerados"  // ¿Hay que borrarlo asi?
      );  // Damos por acabado EventosGenerados

      JU    Final;  // Se ha finalizado


NETWORK
TITLE = Finalizar
// Se acabo la funcion
Final:NOP   0;

END_FUNCTION

FUNCTION "FC803_JDT01EmiJdTMensaje" : Void   // FC803, LAD
TITLE = "EmiJdTMensaje" - Emision de Mensajes
{ S7_Optimized_Access := 'FALSE' }
AUTHOR : TRACKING
NAME : 20141014
VERSION : 4.0
// - Inicializaciones
// - Distrubucion
// - Recoger el Mensaje ACKN
// - Recoger el Mensaje PING o Lista de Eventos
// - Emision del Mensaje
// stored: AutoNumber false, SetENOAutomatically false
   VAR_TEMP
      DBEmiJdT : Word;   // Num. DB de Emision al JdT
      DBUltimoEmi : Word;   // Num. DB del Ultimo Mensaje a Emitir
      DBEmiAK : Word;   // Num. DB del Mensaje AK a Emitir
      Longitud : UDInt;   // Longitud del Mensaje
      CantidadBytes : UDInt;   // Cantidad de Bytes del Mensaje a Enviar
      ReturnValor : Int;   // Temporal
      POrigen : Any;   // Puntero para transferencias y emision
      PDestino : Any;   // Puntero para transferencias
   END_VAR
BEGIN

NETWORK
TITLE = Inicializaciones
// - Inicializa las variables de los DB's
// - Comprueba que el enlace esta activo "EnlaceCP_OK"
// -------------------------------------------------------------------------------------------
// Si trabaja sin Agencia  2018 01 24
      SET;
      AN    "Activar_JDT01";  // Mirar si se trabaja con agencia
      JC    Final;

// ------------------------------------------------------------------------------------------
// Inicializa las variables de los DB's

      L     "JDT1_NDB_EmiMensaje";  // Cogemos el Numero del DB de EmisionMensaje
      T     #DBEmiJdT;
      L     "JDT1_NDB_UltimoEmi";  // Cogemos el Numero del DB de UltimaEmision
      T     #DBUltimoEmi;
      L     "JDT1_NDB_AKEmi";  // Cogemos el Numero del DB de EmisionAK
      T     #DBEmiAK;

// ------------------------------------------------------------------------------------------
// Comprueba el Enlace esta correcto

      A     "DB801_JDT01StatusCOM".EnlaceCP_OK;  // Mirar Si esta el EnlaceCP Activo
      JC    ExisteConexion;  // El EnlaceCP esta OK

// Reseteamos las variables porque El enlaceCP NOK

      R     "DB891_VariablesTCP".TSEND_JdT_PLC_Req;  // Resetear Variables
      R     "DB891_VariablesTCP".TSEND_JdT_PLC_Done;
      R     "DB891_VariablesTCP".TSEND_JdT_PLC_Error;
      R     "DB891_VariablesTCP".TSEND_JdT_PLC_Busy;


      JU    Final;  // Finalizar


NETWORK
TITLE = Distribución
// Hay que seguir este orden:
// - Hay que emitir mensaje
// - Hay que recoger el mensaje ACKN
// - Hay que recoger el mensaje PING o Lista de Eventos
ExisteConexion:NOP   0;

// ------------------------------------------------------------------------------------------
// Hay que emitir mensaje

      L     0;  // Ya tenemos mensaje a Emitir
      LAR1;
      OPN   DB [#DBEmiJdT];
      L     DBB [AR1, P#0.0];
      L     0;
      <>I;
      JC    EmitirMensaje;  // Ir a Emitir

// ------------------------------------------------------------------------------------------
// Hay que recoger Mensaje ACKN para emitir

      L     0;
      LAR1;
      OPN   DB [#DBEmiAK];
      L     DBB [AR1, P#0.0];
      L     2;
      ==I;
      JC    EmitirEvento_AcuseRecibo;  // Ir a Recoger el mensaje AK

// ------------------------------------------------------------------------------------------
// Hay que recoger Mensaje PING o Lista de Eventos para Emitir

      L     0;
      LAR1;
      OPN   DB [#DBUltimoEmi];
      L     DBB [AR1, P#0.0];
      L     2;
      ==I;
      JC    EmitirEvento;  // Ir a Recoger el mensaje KA o de Eventos
      JU    Final;



NETWORK
TITLE = Recoger el Mensaje ACKN - Confirmacion
// Pasos a Seguir:
// - Calcular la Longitud del Mensaje (Puede ser variable)
// - Generamos los punteros Origen y Destino
// - Transferir el Mensaje para Emitir
// - Borrar el Mensaje AK, para decir que lo hemos tratado, y Resetear Variables
// - Emitimos el Mensaje
EmitirEvento_AcuseRecibo:NOP   0;

// ------------------------------------------------------------------------------------------
// 1º Paso - Calcular la longitud del Mensaje

      CALL  "FC890_EtiqChar_EtiqDInt"
      ( DB_String   := "JDT1_NDB_AKEmi",
        Long_String := 5,
        Offset_Ini  := 20,
        Valor       := #Longitud
      );

      L     #Longitud;
      T     #CantidadBytes;

// ------------------------------------------------------------------------------------------
// 2º Paso - Generamos los punteros Origen y Destino

      CALL  "FC897_Generar_PointerAny"
      ( TYP           := 16#10,
        DataTyp       := 16#02,
        repeatcounter := #CantidadBytes,  // Tamaño del mensaje
        DB_Number     := "JDT1_NDB_AKEmi",  // DB donde esta guardado el EmisionAK
        storearea     := 16#84,
        storeaddresse := 16#0000_0000,
        Any_Pointer   := #POrigen  // Puntero del EmisionAK
      );

      CALL  "FC897_Generar_PointerAny"
      ( TYP           := 16#10,
        DataTyp       := 16#02,
        repeatcounter := #CantidadBytes,  // Tamaño del mensaje
        DB_Number     := "JDT1_NDB_EmiMensaje",  // DB donde guardar el EmisionMensaje
        storearea     := 16#84,
        storeaddresse := 16#0000_0000,
        Any_Pointer   := #PDestino  // Puntero del Mensaje a Enviar
      );

// ------------------------------------------------------------------------------------------
// 3º Paso - Transferir en Mensaje para emitir

      CALL  BLKMOV
      ( SRCBLK  := #POrigen,
        RET_VAL := #ReturnValor,
        DSTBLK  := #PDestino
      );

// ------------------------------------------------------------------------------------------
// 4º Paso - Borrar el Mensaje AK y Resetear variables internas

      CALL  "FC898_BorrarMensaje"
      ( DB_A_RESET := "DB806_JDT01EmisionAK"  // ¿Hay que borrar asi?
      );  // Damos por acabado el envio del mensaje

      SET;  // Ya hay Actividad
      R     "DB801_JDT01StatusCOM".SinActividad;

// ------------------------------------------------------------------------------------------
// 5º Paso - Pasamos a Emitir el Mensaje

      L     #CantidadBytes;
      T     "DB801_JDT01StatusCOM".EmiJdT_Longitud;  // Guardamos la longitud para la Emision
      JU    EmitirMensaje;



NETWORK
TITLE = Recoger el Mensaje KA o Lista de Eventos
// Pasos a Seguir:
// - Calcular la Longitud del Mensaje(Puede ser variable)
// - Generamos los punteros Origen y Destino
// - Transferir el Mensaje para Emitir
// - Borrar el Mensaje AK, para decir que lo hemos tratado, y Resetear Variables
// - Emitimos el Mensaje
EmitirEvento:NOP   0;

// ------------------------------------------------------------------------------------------
// 1º Paso - Calcular la longitud del Mensaje

      CALL  "FC890_EtiqChar_EtiqDInt"
      ( DB_String   := "JDT1_NDB_UltimoEmi",
        Long_String := 5,
        Offset_Ini  := 20,
        Valor       := #Longitud
      );

      L     #Longitud;
      T     #CantidadBytes;

// ------------------------------------------------------------------------------------------
// 2º Paso - Generamos los punteros Origen y Destino

      CALL  "FC897_Generar_PointerAny"
      ( TYP           := 16#10,
        DataTyp       := 16#02,
        repeatcounter := #CantidadBytes,  // Tamaño del mensaje
        DB_Number     := "JDT1_NDB_UltimoEmi",  // DB donde esta guardado el UltimoMensaje
        storearea     := 16#84,
        storeaddresse := 16#0000_0000,
        Any_Pointer   := #POrigen  // Puntero del UltimoMensaje
      );

      CALL  "FC897_Generar_PointerAny"
      ( TYP           := 16#10,
        DataTyp       := 16#02,
        repeatcounter := #CantidadBytes,  // Tamaño del mensaje
        DB_Number     := "JDT1_NDB_EmiMensaje",  // DB donde guardar el Emisio del Mensaje
        storearea     := 16#84,
        storeaddresse := 16#0000_0000,
        Any_Pointer   := #PDestino  // Puntero del Mensaje a Enviar
      );

// ------------------------------------------------------------------------------------------
// 3º Paso - Transferir

      CALL  BLKMOV
      ( SRCBLK  := #POrigen,
        RET_VAL := #ReturnValor,
        DSTBLK  := #PDestino
      );

// ------------------------------------------------------------------------------------------
// 4º Paso - Borrar el Mensaje Tratado y Resetear variables internas

      SET;  // Ya hay Actividad
      R     "DB801_JDT01StatusCOM".SinActividad;

// Parar Borrar el Mensaje hay que saber de que tipo es:
// KA o Lista de Eventos - Porque se hace cosas diferentes

      L     0;
      LAR1;
      OPN   DB [#DBUltimoEmi];
      L     DBD [AR1, P#24.0];
      L     'PING';
      <>I;
      JC    _040;  // Si no es KA hay que borrarlo entero

// Es Mensaje KA - Borrar todo el Mensaje
      CALL  "FC898_BorrarMensaje"
      ( DB_A_RESET := "DB805_JDT01UltimoEnviado"  // ¿Hay que borrar asi?
      );  // Damos por acabado el envio del mensaje KA

      JU    _041;

// Es Mnesaje de Lista de Eventos lo damos por tratado
_040: OPN   DB [#DBUltimoEmi];  // Damos por enviado el mensaje de Evento
      L     'N';
      T     DBB [AR1, P#0.0];

      JU    _041;

// ------------------------------------------------------------------------------------------
// 5º Paso - Pasamos a Emitir el Mensaje

_041: L     #CantidadBytes;
      T     "DB801_JDT01StatusCOM".EmiJdT_Longitud;  // Guardamos la longitud para la Emision
      JU    EmitirMensaje;



NETWORK
TITLE = Emision del Mensaje
// Pasos a Seguir
// - Control de la Emision
// - Calcular el puntero de lo que tenemos que emitir
// - Emision del Mensaje
// - Comprobacion del Mensaje Enviado
EmitirMensaje:NOP   0;

// ------------------------------------------------------------------------------------------
// 1º Paso - Control de la Emision

      AN    "DB891_VariablesTCP".TSEND_JdT_PLC_Busy;
      AN    "DB891_VariablesTCP".TSEND_JdT_PLC_Req;
      AN    "DB891_VariablesTCP".TSEND_JdT_PLC_Flanco;
      =     "DB891_VariablesTCP".TSEND_JdT_PLC_Flanco;

      A     "DB891_VariablesTCP".TSEND_JdT_PLC_Flanco;
      AN    "DB891_VariablesTCP".TSEND_JdT_PLC_Req;
      S     "DB891_VariablesTCP".TSEND_JdT_PLC_Req;


// ------------------------------------------------------------------------------------------
// 2º Paso - Generar el Puntero de lo que se tiene que Emitir

      CALL  "FC897_Generar_PointerAny"
      ( TYP           := 16#10,
        DataTyp       := 16#02,
        repeatcounter := "DB801_JDT01StatusCOM".EmiJdT_Longitud,  // Tamaño del mensaje
        DB_Number     := "JDT1_NDB_EmiMensaje",  // DB donde esta guardado el EmisionMensaje
        storearea     := 16#84,
        storeaddresse := 16#0000_0000,
        Any_Pointer   := #POrigen  // Puntero del EmisionMensaje
      );

// ------------------------------------------------------------------------------------------
// 2º Paso - Emision del Mensaje

      CALL  TSEND, "DB894_TSEND_JdT_PLC"
      ( REQ    := "DB891_VariablesTCP".TSEND_JdT_PLC_Flanco,
        ID     := W#16#1,
        LEN    := "DB801_JDT01StatusCOM".EmiJdT_Longitud,
        DONE   := "DB891_VariablesTCP".TSEND_JdT_PLC_Done,
        BUSY   := "DB891_VariablesTCP".TSEND_JdT_PLC_Busy,
        ERROR  := "DB891_VariablesTCP".TSEND_JdT_PLC_Error,
        STATUS := "DB891_VariablesTCP".TSEND_JdT_PLC_Status,
        DATA   := #POrigen
      );


// ------------------------------------------------------------------------------------------
// 3º Paso - Comprobacion del Mensaje Enviado

      A     "DB891_VariablesTCP".TSEND_JdT_PLC_Req;  // Si llega Error en la Emision
      AN    "DB891_VariablesTCP".TSEND_JdT_PLC_Done;  // Restear
      A     "DB891_VariablesTCP".TSEND_JdT_PLC_Error;
      S     "DB801_JDT01StatusCOM".EmiJdT_Reset;
      R     "DB891_VariablesTCP".TSEND_JdT_PLC_Req;

